// TwinCAT 3 PLC project PRG_PLC
// ProgramVersion: 3.1.4023.0
// CompilerDefines: VISU_USEWSTRING
// libraries:
//   Tc2_Standard, * (Beckhoff Automation GmbH)
//   Tc2_System, * (Beckhoff Automation GmbH)
//   Tc2_Utilities, * (Beckhoff Automation GmbH)
//   Tc3_Module, * (Beckhoff Automation GmbH)
//   VisuDialogs, * (System)
//   VisuSymbols,3.5.10.0,System
// project tree:
//   / GlobalTextList.TcGTLO, ImagePool.TcIPO (not stored), PlcTask.TcTTO, Visualization Manager.TcVMO (not stored), VISU_TASK.TcTTO
//   GVLs/ GVL_Elementy.TcGVL, GVL_Parametry.TcGVL, GVL_Podzespoly.TcGVL, GVL_Wejscia_IO.TcGVL, GVL_Wyjscia_IO.TcGVL
//   POUs/01 - Elementy/Czujnik/ITF/ ITF_Czujnik.TcIO
//   POUs/01 - Elementy/Czujnik/POU/ FB_Czujnik_NC.TcPOU, FB_Czujnik_NO.TcPOU
//   POUs/01 - Elementy/Elektrozawór/ITF/ ITF_Elektozawor.TcIO
//   POUs/01 - Elementy/Elektrozawór/POU/ FB_Elektrozawor_5na2_1Cewka.TcPOU, FB_Elektrozawor_5na2_2Cewki.TcPOU, FB_Elektrozawor_5na3_Odpowietrzony.TcPOU, FB_Elektrozawor_5na3_Zapowietrzony.TcPOU
//   POUs/01 - Elementy/Silownik/DUT/ DUT_SilownikParametry.TcDUT
//   POUs/01 - Elementy/Silownik/ITF/ ITF_Silownik.TcIO
//   POUs/01 - Elementy/Silownik/POU/ FB_Silownik.TcPOU, FB_Silownik_Kontrola.TcPOU, FB_Silownik_Kontrola_Komunikacja.TcPOU
//   POUs/02 - Przesuwacz Na Silowniku/DUT/ DUT_PrzesuwaczNaSilowniku_Parametry.TcDUT (not stored)
//   POUs/02 - Przesuwacz Na Silowniku/POU/ FB_PrzesuwaczNaSilowniku.TcPOU, FB_PrzesuwaczNaSilowniku_Komunikacja.TcPOU (not stored)
//   POUs/03 - Ciecie/DUT/ DUT_Ciecie_Parametry.TcDUT
//   POUs/03 - Ciecie/POU/ FB_Ciecie.TcPOU, FB_Ciecie_Komunikacja.TcPOU
//   POUs/50 - testowy podzespol/POU/ FB_TestowyPodzespol.TcPOU
//   POUs/51 - Krajalnica/DUT/ DUT_Krajalnica_Parametry.TcDUT, DUT_Krajalnica_StanyPodzespolow.TcDUT, DUT_Krajalnica_Symulacja.TcDUT
//   POUs/51 - Krajalnica/POU/ FB_Krajalnica.TcPOU, FB_Krajalnica_Komunikacja.TcPOU
//   POUs/80 - Symulacja pracy/DUT/ DUT_Symulacja_Parametry.TcDUT
//   POUs/80 - Symulacja pracy/POU/ FB_Symulacja.TcPOU
//   POUs/90 - Stan Maszyny/DUT/ DUT_StanMaszyny_VISU_Stan.TcDUT, E_PMLState.TcDUT, E_PMLUnitMode.TcDUT
//   POUs/90 - Stan Maszyny/GVL/ GVL_StanMaszyny.TcGVL, GVL_StanMaszyny_STALE.TcGVL
//   POUs/90 - Stan Maszyny/ITF/ ITF_StanMaszyny.TcIO
//   POUs/90 - Stan Maszyny/POU/ FB_StanMaszyny.TcPOU, FB_StanMaszyny_Baza.TcPOU
//   POUs/90 - Stan Maszyny/Visu/ Visu_StanMaszyny_AktualyStan.TcVIS, Visu_StanMaszyny_AktualyStan_BezNaciskania.TcVIS, Visu_StanMaszyny_Diagram.TcVIS, Visu_StanMaszyny_DiagramZPrzyciskami.TcVIS
//   POUs/91 - Elementy Sterujace/GVL/ GVL_ElementySterujace.TcGVL
//   POUs/91 - Elementy Sterujace/POU/ FB_ElementySterujace.TcPOU
//   POUs/92 - Elementy maszyny/Impulsy/POU/ FB_Impulsy.TcPOU
//   POUs/92 - Elementy maszyny/Przycisk/ITF/ ITF_Przycisk.TcIO
//   POUs/92 - Elementy maszyny/Przycisk/POU/ FB_Przycisk_NC.TcPOU, FB_Przycisk_NO.TcPOU
//   POUs/92 - Elementy maszyny/Wieza Sygnalizacyjna/ITF/ ITF_WiezaSygnalizacyjna.TcIO
//   POUs/92 - Elementy maszyny/Wieza Sygnalizacyjna/POU/ FB_WiezaSygnalizacyjna_Cyfrowe.TcPOU
//   POUs/93 - Podzespol/ITF/ ITF_Podzespol.TcIO
//   POUs/93 - Podzespol/POU/ FB_Podzespol.TcPOU
//   POUs/95 - Logowanie bledow/DUT/ DUT_LogowanieBledow_WyswietlanieParametry.TcDUT, DUT_LogowanieBledow_Zapamietanych.TcDUT, DUT_LogowanieBledow_Zdarzenie.TcDUT, DUT_LogowanieBledow_ZdarzenieOpis.TcDUT, DUT_LogowanieBledow_ZdarzenieStan.TcDUT, DUT_LogowanieBledow_ZdarzenieWyswietlane.TcDUT
//   POUs/95 - Logowanie bledow/GVL/ GVL_LogowanieBledow.TcGVL, GVL_LogowanieBledow_Stale.TcGVL
//   POUs/95 - Logowanie bledow/ITF/ ITF_LogowanieBledow_ElementWykonawczy.TcIO
//   POUs/95 - Logowanie bledow/POU/ FB_LogowanieBledow.TcPOU, FB_LogowanieBledow_ElementWykonawczy.TcPOU, FB_LogowanieBledow_ElementZlozony.TcPOU
//   POUs/95 - Logowanie bledow/Wizualizacja/ Visu_LogowanieBledow_Tabela.TcVIS
//   POUs/99 - Wizualizacja/DUT/ DUT_Wizualizacja_SymulacjaDane.TcDUT
//   POUs/99 - Wizualizacja/GVL/ GVL_Wizualizacja.TcGVL (not stored)
//   POUs/99 - Wizualizacja/POU/ FB_Wizualizacja.TcPOU
//   POUs/ MAIN.TcPOU
//   VISUs/ OknoGlowne.TcVIS, Symulacja.TcVIS, Ustawienia.TcVIS, Visualization.TcVIS
// real-time tasks:
//   TASK PlcTask: cycle T#10ms, priority 20, ADS port 350
//   TASK VISU_TASK: cycle T#200000us, priority 30, ADS port 351

CONFIGURATION PRG_PLC
    RESOURCE PLC ON TwinCAT3
        TASK PlcTask(INTERVAL := T#10ms, PRIORITY := 20);
        TASK VISU_TASK(INTERVAL := T#100us, PRIORITY := 30);
        PROGRAM MAIN WITH PlcTask : MAIN;
        PROGRAM VisuElems_Visu_Prg WITH VISU_TASK : VisuElems.Visu_Prg;
    END_RESOURCE
END_CONFIGURATION

// ---- POUs/01 - Elementy/Silownik/DUT/DUT_SilownikParametry.TcDUT
TYPE DUT_SilownikParametry :
STRUCT
	rCzasNaPrace							: REAL := 5000;
	rCzasNaPowrot							: REAL := 5000;
END_STRUCT
END_TYPE

// ---- POUs/03 - Ciecie/DUT/DUT_Ciecie_Parametry.TcDUT
TYPE DUT_Ciecie_Parametry :
STRUCT
	stNaped									: DUT_SilownikParametry;
	rOdczekaj								: real := 1000; 	//chwila na odczekanie po cięciu
END_STRUCT
END_TYPE

// ---- POUs/51 - Krajalnica/DUT/DUT_Krajalnica_Parametry.TcDUT
TYPE DUT_Krajalnica_Parametry :
STRUCT
	stCiecie1								: DUT_Ciecie_Parametry;	
	stCiecie2								: DUT_Ciecie_Parametry;
	stPodawanieWafla						: DUT_PrzesuwaczNaSilowniku_Parametry;
	
	
END_STRUCT
END_TYPE

// ---- POUs/51 - Krajalnica/DUT/DUT_Krajalnica_StanyPodzespolow.TcDUT
TYPE DUT_Krajalnica_StanyPodzespolow :
STRUCT
	bCiecie1_Bazowanie						: BOOL;
	bCiecie1_Ciecie							: BOOL;
	bCiecie1_Naped_WStronePoczatku			: BOOL;
	bCiecie1_Naped_WStroneKonca				: BOOL;			

	bCiecie2_Bazowanie						: BOOL;
	bCiecie2_Ciecie							: BOOL;
	bCiecie2_Naped_WStronePoczatku			: BOOL;
	bCiecie2_Naped_WStroneKonca				: BOOL;			

	bPodawanie_Bazowanie					: BOOL;
	bPodawanie_Podawanie					: BOOL;
	bPodawanie_Zabierak_WStronePoczatku		: BOOL;
	bPodawanie_zabierak_WStroneKonca		: BOOL;
	bPodawanie_Przesuwanie_WStronePoczatku	: BOOL;
	bPodawanie_Przesuwanie_WStroneKonca		: BOOL;

	
END_STRUCT
END_TYPE

// ---- POUs/51 - Krajalnica/DUT/DUT_Krajalnica_Symulacja.TcDUT
TYPE DUT_Krajalnica_Symulacja :
STRUCT
	bCiecie1Bazuj							: BOOL;		
	bCiecie1Tnij							: BOOL;
	bCiecie2Bazuj							: BOOL;		
	bCiecie2Tnij							: BOOL;
	bPodawanieBazuj							: BOOL;		
	bPodawaniePodaj							: BOOL;	
	
END_STRUCT
END_TYPE

// ---- POUs/80 - Symulacja pracy/DUT/DUT_Symulacja_Parametry.TcDUT
TYPE DUT_Symulacja_Parametry :
STRUCT
	rCiecie1_BazowanieCzasNaPowrot			: REAL := 2000;
	rCiecie1_CiecieCzasNaCiecie				: REAL := 2000;
	rCiecie1_CiecieCzasNaPowrot				: REAL := 2000;
	
	rCiecie2_BazowanieCzasNaPowrot			: REAL := 2000;
	rCiecie2_CiecieCzasNaCiecie				: REAL := 2000;
	rCiecie2_CiecieCzasNaPowrot				: REAL := 2000;
	
	rPodawanieZabierak_BazowanieCzasNaPowrot	: REAL := 1000;
	rPodawaniePrzesuwanie_BazowanieCzasNaPowrot	: REAL := 2000;
	
	rPodawanieZabierak_PodawanieCzasNaPrace			: REAL := 1000;
	rPodawanieZabierak_PodawanieCzasNaPowrot		: REAL := 1000;
	rPodawaniePrzesuwanie_PodawanieCzasNaPobranie	: REAL := 2000;
	rPodawaniePrzesuwanie_PodawanieCzasNaPodanie	: REAL := 2000;
	
END_STRUCT
END_TYPE

// ---- POUs/90 - Stan Maszyny/DUT/DUT_StanMaszyny_VISU_Stan.TcDUT
//==================================================================================================
//								RJM Maszyny sp. z o.o.
//									27.06.2022
//	Struktura sterująca wyświetlania pojedynczego stanu
// 	v1.0	|| TC v 3.1.4024.29		|| - pierwsza wersja
//==================================================================================================
TYPE DUT_StanMaszyny_VISU_Stan :
STRUCT
	bAktywny								: BOOL;
	sNazwa									: STRING;
	dwKolorTla								: DWORD;
	bWygaszone								: BOOL;
END_STRUCT
END_TYPE

// ---- POUs/90 - Stan Maszyny/DUT/E_PMLState.TcDUT
(* states according to PackTags v3.0 *)
//==================================================================================================
//								RJM Maszyny sp. z o.o.
//									27.06.2022
//	Spis dostepnych stanow maszyny
// 	v1.0	|| TC v 3.1.4024.29		|| - pierwsza wersja
//==================================================================================================
{attribute 'qualified_only'}
{attribute 'strict'}
TYPE E_PMLState :
(
	UNDEFINED		:=  0,
	CLEARING 		:=  1,
	STOPPED 		:=  2,
	STARTING 		:=  3,
	IDLE 			:=  4,
	SUSPENDED 		:=  5,
	EXECUTE 		:=  6,
	STOPPING	 	:=  7,
	ABORTING 		:=  8,
	ABORTED 		:=  9,
	HOLDING 		:= 10,
	HELD 			:= 11,
	UNHOLDING 		:= 12,
	SUSPENDING 		:= 13,
	UNSUSPENDING 	:= 14,
	RESETTING 		:= 15,
	COMPLETING 		:= 16,
	COMPLETE	 	:= 17
);
END_TYPE

// ---- POUs/90 - Stan Maszyny/DUT/E_PMLUnitMode.TcDUT
{attribute 'qualified_only'}
{attribute 'strict'}
//==================================================================================================
//								RJM Maszyny sp. z o.o.
//									27.06.2022
//	Spis dostepnych trybow pracy maszyny
// 	v1.0	|| TC v 3.1.4024.29		|| - pierwsza wersja
//==================================================================================================
TYPE E_PMLUnitMode :
(
	UNDEFINED		:=  0,
	AUTOMATIC		:=  1,
	MAINTENANCE 	:=  2,
	MANUAL 			:=  3,
	SEMIAUTOMATIC	:=  4,
	DRYRUN			:=  5,
	USERMODE1		:=  6,
	USERMODE2		:=  7,
	IDLE 			:=  8,
	ESTOP 			:=  9
);
END_TYPE

// ---- POUs/95 - Logowanie bledow/DUT/DUT_LogowanieBledow_WyswietlanieParametry.TcDUT
//==================================================================================================
//								RJM Maszyny sp. z o.o.
//									04.02.2022
//	Struktura parametrów wyświetlania danych historii zdarzeń
// 	v1.0	|| TC v 3.1.4024.22		|| - pierwsza wersja
//==================================================================================================
TYPE DUT_LogowanieBledow_WyswietlanieParametry :
STRUCT
//FILTRY WYSIETLANIA
	// Flagi wykonywalnosci
	bFiltrID								: BOOL;
	bFiltrRodzaj							: BOOL;
	bFiltrStartOD							: BOOL;
	bFiltrStartDO							: BOOL;
	bFiltrKoniecOD							: BOOL;
	bFiltrKoniecDO							: BOOL;
	bFiltrAktywne							: BOOL;
	// Parametry
	iFiltrID								: INT;	
	byFiltrRodzaj							: BYTE;
	dtFiltrStartOD							: DT;
	dtFiltrStartDO							: DT;
	dtFiltrKoniecOD							: DT;
	dtFiltrKoniecDO							: DT;
	
END_STRUCT
END_TYPE

// ---- POUs/95 - Logowanie bledow/DUT/DUT_LogowanieBledow_Zapamietanych.TcDUT
TYPE DUT_LogowanieBledow_Zapamietanych :
STRUCT
	iIdZdarzenia							: INT;
	dtDataStart								: DT;
	dtDataKoniec							: DT;
	bAktywne								: BOOL;
END_STRUCT
END_TYPE

// ---- POUs/95 - Logowanie bledow/DUT/DUT_LogowanieBledow_Zdarzenie.TcDUT
TYPE DUT_LogowanieBledow_Zdarzenie :
STRUCT
	iIdZdarzenia							: INT;
	sNrKomponentu							: STRING[10];
	sKodBledu								: STRING[10];
	byRodzajZdarzenia						: BYTE;	//1 - blad, 2 - ostrzezenie, 3 - wiadomosc, 4 - safety
END_STRUCT
END_TYPE

// ---- POUs/95 - Logowanie bledow/DUT/DUT_LogowanieBledow_ZdarzenieOpis.TcDUT
TYPE DUT_LogowanieBledow_ZdarzenieOpis :
STRUCT
	iIdZdarzenia							: INT;
	sOpis									: STRING;
END_STRUCT
END_TYPE

// ---- POUs/95 - Logowanie bledow/DUT/DUT_LogowanieBledow_ZdarzenieStan.TcDUT
TYPE DUT_LogowanieBledow_ZdarzenieStan :
STRUCT
	iIdZdarzenia							: INT;
	bAktywne								: BOOL;
END_STRUCT
END_TYPE

// ---- POUs/95 - Logowanie bledow/DUT/DUT_LogowanieBledow_ZdarzenieWyswietlane.TcDUT
TYPE DUT_LogowanieBledow_ZdarzenieWyswietlane :
STRUCT
	sNrKomponentu							: STRING[10];
	sKodBledu								: STRING[10];
	byRodzajZdarzenia						: BYTE;
	sOpis									: STRING;
	dtDataStart								: DT;
	dtDataKoniec							: DT;
	dwKolor									: UDINT;
END_STRUCT
END_TYPE

// ---- POUs/99 - Wizualizacja/DUT/DUT_Wizualizacja_SymulacjaDane.TcDUT
TYPE DUT_Wizualizacja_SymulacjaDane :
STRUCT
	stStanySilownikow						: DUT_Krajalnica_StanyPodzespolow;
	eTrybPracy								: E_PMLUnitMode;
	bCiecie1_Poczatek						: BOOL;
	bCiecie1_Koniec							: BOOL;
	bCiecie2_Poczatek						: BOOL;
	bCiecie2_Koniec							: BOOL;
	bPodawanieZabierakPoczatek				: BOOL;
	bPodawanieZabierakKoniec				: BOOL;
	bPodawaniePrzesuwaniePoczatek			: BOOL;
	bPodawaniePrzesuwanieKoniec				: BOOL;
	bCzujnikWaflaDoPodania					: BOOL;
	bCzujnikWaflaDoCiecia1					: BOOL;
	bCzujnikWaflaDoCiecia2					: BOOL;	
	
	bCiecie1Bazuj							: BOOL;
	bCiecie1Tnij							: BOOL;
	bCiecie2Bazuj							: BOOL;		
	bCiecie2Tnij							: BOOL;
	bPodawanieBazuj							: BOOL;		
	bPodawaniePodaj							: BOOL;	

END_STRUCT
END_TYPE

// ---- GVLs/GVL_Elementy.TcGVL
{attribute 'qualified_only'}
{attribute 'global_init_slot' := '40501'}
VAR_GLOBAL
	fbPrzysciskStart						: FB_Przycisk_NO;
	fbPrzyciskStop							: FB_Przycisk_NO;
	fbWieza									: FB_WiezaSygnalizacyjna_Cyfrowe;

END_VAR



	(*
	fbSilownikCiecia1						: FB_Silownik_Kontrola (	fbCzujnikPozycja0 			:= GVL_Wejscia_IO.bCzujnik0C1, 
																		fbCzujnikPozycjaMax 		:= GVL_Wejscia_IO.bCzujnikMaxC1,
																		fbElektrozawor 				:= GVL_Wyjscia_IO.fbElektrozaworC1);

	fbSilownikCiecia2						: FB_Silownik_Kontrola (	fbCzujnikPozycja0 			:= GVL_Wejscia_IO.bCzujnik0C2, 
																		fbCzujnikPozycjaMax 		:= GVL_Wejscia_IO.bCzujnikMaxC2,
																		fbElektrozawor 				:= GVL_Wyjscia_IO.fbElektrozaworC2);

	fbPodawanieWaflaZabierak				: FB_Silownik_Kontrola (	fbCzujnikPozycja0 			:= GVL_Wejscia_IO.bCzujnik0PW_Z, 
																		fbCzujnikPozycjaMax 		:= GVL_Wejscia_IO.bCzujnikMaxPW_Z,
																		fbElektrozawor 				:= GVL_Wyjscia_IO.fbElektrozaworPW_Z);																	
		
	fbPodawanieWaflaPrzesuwanie				: FB_Silownik_Kontrola (	fbCzujnikPozycja0 			:= GVL_Wejscia_IO.bCzujnik0PW_N, 
																		fbCzujnikPozycjaMax 		:= GVL_Wejscia_IO.bCzujnikMaxPW_N,
																		fbElektrozawor 				:= GVL_Wyjscia_IO.fbElektrozaworPW_N);																	

	*)

// ---- GVLs/GVL_Parametry.TcGVL
{attribute 'qualified_only'}
VAR_GLOBAL
	stSymulacja								: DUT_Symulacja_Parametry;
	stKrajalnica							: DUT_Krajalnica_Parametry;
END_VAR

// ---- GVLs/GVL_Podzespoly.TcGVL
{attribute 'qualified_only'}
{attribute 'global_init_slot' := '40505'}
VAR_GLOBAL
	
	fbSymulacja								: FB_Symulacja;	

	fbKrajalnica							: FB_Krajalnica ( 	bC1_Czujnik0					:= GVL_Wejscia_IO.bCzujnik0C1,	
                                                                bC1_CzujnikMax					:= GVL_Wejscia_IO.bCzujnikMaxC1,
                                                                fbC1_Elektrozawor				:= GVL_Wyjscia_IO.fbElektrozaworC1,
																bC2_Czujnik0					:= GVL_Wejscia_IO.bCzujnik0C2,	
                                                                bC2_CzujnikMax					:= GVL_Wejscia_IO.bCzujnikMaxC2,
                                                                fbC2_Elektrozawor				:= GVL_Wyjscia_IO.fbElektrozaworC2,
																bPW_Z_Czujnik0		    		:= GVL_Wejscia_IO.bCzujnik0PW_Z,
																bPW_Z_CzujnikMax	   			:= GVL_Wejscia_IO.bCzujnikMaxPW_Z,
																fbPW_Z_Elektrozawor				:= GVL_Wyjscia_IO.fbElektrozaworPW_Z,
																bPW_P_Czujnik0		    		:= GVL_Wejscia_IO.bCzujnik0PW_N,
																bPW_P_CzujnikMax	   			:= GVL_Wejscia_IO.bCzujnikMaxPW_N,
																fbPW_P_Elektrozawor				:= GVL_Wyjscia_IO.fbElektrozaworPW_N,
																bWafalNaWejsciu					:= GVL_Wejscia_IO.bWafelNaWejsciu,
                                                                bWafalDoCiecia1					:= GVL_Wejscia_IO.bWafelDoCiecia1,
                                                                bWafalDoCiecia2					:= GVL_Wejscia_IO.bWafelDoCiecia2);

															
END_VAR

// ---- GVLs/GVL_Wejscia_IO.TcGVL
{attribute 'qualified_only'}
{attribute 'global_init_slot' := '40501'}
VAR_GLOBAL
//Przyciski	
	
//czujniki siłownika ciecia 1
	bCzujnik0C1								: FB_Czujnik_NO;
	bCzujnikMaxC1							: FB_Czujnik_NO;
//czujniki siłownika ciecia 2
	bCzujnik0C2								: FB_Czujnik_NO;
	bCzujnikMaxC2							: FB_Czujnik_NO;
//czujniki przesuwacza wafla
	bCzujnik0PW_Z							: FB_Czujnik_NO;
	bCzujnikMaxPW_Z							: FB_Czujnik_NO;
	bCzujnik0PW_N							: FB_Czujnik_NO;
	bCzujnikMaxPW_N							: FB_Czujnik_NO;
//czujnik waflae
	bWafelNaWejsciu							: FB_Czujnik_NO;
	bWafelDoCiecia1							: FB_Czujnik_NO;
	bWafelDoCiecia2							: FB_Czujnik_NO;
	
END_VAR

// ---- GVLs/GVL_Wyjscia_IO.TcGVL
{attribute 'qualified_only'}
{attribute 'global_init_slot' := '40510'}
VAR_GLOBAL
//elektrozawor siłownika 1
	fbElektrozaworC1						: FB_Elektrozawor_5na2_2Cewki;
//elektrozawor siłownika 2
	fbElektrozaworC2						: FB_Elektrozawor_5na2_2Cewki;
//elektrozawory przesuwacza
	fbElektrozaworPW_Z						: FB_Elektrozawor_5na2_2Cewki;
	fbElektrozaworPW_N						: FB_Elektrozawor_5na2_2Cewki;
END_VAR

// ---- POUs/90 - Stan Maszyny/GVL/GVL_StanMaszyny.TcGVL
{attribute 'qualified_only'}
{attribute 'global_init_slot' := '40515'}
VAR_GLOBAL

	arrPodzesoly							: ARRAY [1..GVL_StanMaszyny_Stale.MAX_LICZBA_PODZESPOLOW] OF ITF_StanMaszyny :=[
																GVL_Podzespoly.fbSymulacja,
																GVL_Podzespoly.fbKrajalnica];
	fbStanMaszyny							: FB_StanMaszyny (arrPodzesoly := arrPodzesoly,
																iIloscDodanychPodzespolow := 2);
	bStart									: BOOL;
	bStop									: BOOL;
	bReset									: BOOL;
	bAbort									: BOOL;
	bClear									: BOOL;
	bHold									: BOOL;
	bUnhold									: BOOL;
	bSuspend								: BOOL;
	bUnsuspend								: BOOL;
	eTrybPracy								: E_PMLUnitMode := E_PMLUnitMode.MANUAL;		
	bWlaczPrzyciski							: BOOL;												
	
END_VAR

// ---- POUs/90 - Stan Maszyny/GVL/GVL_StanMaszyny_STALE.TcGVL
{attribute 'qualified_only'}
VAR_GLOBAL CONSTANT
	MAX_LICZBA_PODZESPOLOW					: int := 10;
END_VAR

// ---- POUs/91 - Elementy Sterujace/GVL/GVL_ElementySterujace.TcGVL
{attribute 'qualified_only'}
{attribute 'global_init_slot' := '40520'}
VAR_GLOBAL
	fbElementySterujace						: FB_ElementySterujace (
													fbWieza					:= GVL_Elementy.fbWieza,
													fbPrzyciskStart			:= GVL_Elementy.fbPrzysciskStart,
													fbPrzyciskStop			:= GVL_Elementy.fbPrzyciskStop
												);
												
END_VAR

// ---- POUs/95 - Logowanie bledow/GVL/GVL_LogowanieBledow.TcGVL
{attribute 'qualified_only'}
{attribute 'global_init_slot' := '40550'}
VAR_GLOBAL
	arrElementyWykonawcze 					: ARRAY [1..GVL_LogowanieBledow_Stale.MAX_ILOSC_ELEMENTOW] OF 
																ITF_LogowanieBledow_ElementWykonawczy := [
																	GVL_Podzespoly.fbKrajalnica.fbLBKomunikacja];

	fbLoger 								: FB_LogowanieBledow (	tablica := arrElementyWykonawcze,
																	iIloscDodanychElementow := 1);
	bWyswietlAlarmy							: BOOL;																
	
END_VAR
VAR_GLOBAL //PERSISTENT
	arrTablicaZdarzenZapamietancyh			: ARRAY [1..GVL_LogowanieBledow_Stale.MAX_ILOSC_ZDARZEN_ZAPAMIETANYCH] OF DUT_LogowanieBledow_Zapamietanych;																
	
	iIloscZdarzenZapamietanych				: INT;	//ilosc zdarzen ktore wystapiły
END_VAR

// ---- POUs/95 - Logowanie bledow/GVL/GVL_LogowanieBledow_Stale.TcGVL
{attribute 'qualified_only'}
VAR_GLOBAL CONSTANT
	MAX_ILOSC_ELEMENTOW						: INT := 10;	//Ilosc elementow zlozonych
	MAX_ILOSC_ZDARZEN_NA_ELEMENT			: INT := 10;	//ilosc zdarzen na element
	MAX_ILOSC_ELEMENTOW_NA_PODZESPOL		: INT := 10;	//Ilosc elementow na element złozony
	MAX_ILOSC_ZDARZEN						: INT := 100;	//ilosc zdarzen zdefiniowanych
	MAX_ILOSC_ZDARZEN_DO_WYSWIETLANIA		: INT := 50;	//ilosc wyswietlanych zdarzen z tablicy zapamietanych
	MAX_ILOSC_ZDARZEN_ZAPAMIETANYCH			: INT := 200;	//ilosc zadarzen zapamietanych
END_VAR

// ---- POUs/01 - Elementy/Czujnik/ITF/ITF_Czujnik.TcIO
//==================================================================================================
//								RJM Maszyny sp. z o.o.
//									04.06.2022
//	Obsługa czujnika  
// 	v1.0	|| TC v 3.1.4024.22		|| - pierwsza wersja
//==================================================================================================
INTERFACE ITF_Czujnik

//==================================================================================================
//								RJM Maszyny sp. z o.o.
//									13.05.2022
//	Informacja czy czujnik jest zadziałany 
// 	v1.0	|| TC v 3.1.4024.22		|| - pierwsza wersja
//==================================================================================================
PROPERTY CzyZadzialany : BOOL
GET
END_GET
END_PROPERTY

END_INTERFACE

// ---- POUs/01 - Elementy/Elektrozawór/ITF/ITF_Elektozawor.TcIO
//==================================================================================================
//								RJM Maszyny sp. z o.o.
//									04.06.2022
//	Sterowanie elektrozaworem  
// 	v1.0	|| TC v 3.1.4024.22		|| - pierwsza wersja
//==================================================================================================
INTERFACE ITF_Elektozawor

//==================================================================================================
//								RJM Maszyny sp. z o.o.
//									04.06.2022
//	Sterowanie cewkami elektrozaworu 
// 	v1.0	|| TC v 3.1.4024.22		|| - pierwsza wersja
//==================================================================================================
METHOD Steruj : BOOL
VAR_INPUT
	bKierunekWstrone0						: BOOL;
	bKierunekWStroneMax						: BOOL;	
END_VAR
END_METHOD

END_INTERFACE

// ---- POUs/01 - Elementy/Silownik/ITF/ITF_Silownik.TcIO
//==================================================================================================
//								RJM Maszyny sp. z o.o.
//									13.05.2022
//	Obsługa silonwika
// 	v1.0	|| TC v 3.1.4024.22		|| - pierwsza wersja
//==================================================================================================
INTERFACE ITF_Silownik

//==================================================================================================
//								RJM Maszyny sp. z o.o.
//									13.05.2022
//	Informaca czy  tłoczysko jest na końca
// 	v1.0	|| TC v 3.1.4024.22		|| - pierwsza wersja
//==================================================================================================
PROPERTY NaKoncu : BOOL
GET
END_GET
END_PROPERTY

//==================================================================================================
//								RJM Maszyny sp. z o.o.
//									13.05.2022
//	Informaca czy  tłoczysko jest na poczatku
// 	v1.0	|| TC v 3.1.4024.22		|| - pierwsza wersja
//==================================================================================================
PROPERTY NaPoczatku : BOOL
GET
END_GET
END_PROPERTY

//==================================================================================================
//								RJM Maszyny sp. z o.o.
//									13.05.2022
//	Przesun tłoczysko w strone końca
// 	v1.0	|| TC v 3.1.4024.22		|| - pierwsza wersja
//==================================================================================================
PROPERTY PrzesunDoKonca : BOOL
SET
END_SET
END_PROPERTY

//==================================================================================================
//								RJM Maszyny sp. z o.o.
//									13.05.2022
//	Przesun tłoczysko w strone poczatku
// 	v1.0	|| TC v 3.1.4024.22		|| - pierwsza wersja
//==================================================================================================
PROPERTY PrzesunDoPoczatku : BOOL
SET
END_SET
END_PROPERTY

//==================================================================================================
//								RJM Maszyny sp. z o.o.
//									13.05.2022
//	Przesuwanie tłoczyska w strone końca
// 	v1.0	|| TC v 3.1.4024.22		|| - pierwsza wersja
//==================================================================================================
PROPERTY PrzesuwanieWStroneKonca : BOOL
GET
END_GET
END_PROPERTY

//==================================================================================================
//								RJM Maszyny sp. z o.o.
//									13.05.2022
//	Przesuwanie tłoczyska w strone poczatku
// 	v1.0	|| TC v 3.1.4024.22		|| - pierwsza wersja
//==================================================================================================
PROPERTY PrzesuwanieWStronePoczatku : BOOL
GET
END_GET
END_PROPERTY

END_INTERFACE

// ---- POUs/90 - Stan Maszyny/ITF/ITF_StanMaszyny.TcIO
INTERFACE ITF_StanMaszyny

//==================================================================================================
//								RJM Maszyny sp. z o.o.
//									5.06.2022
//	Stan maszyny Aborted - metoda pusta
// 	v1.0	|| TC v 3.1.4024.29		|| - pierwsza wersja
//==================================================================================================
METHOD SM_Aborted : BOOL
VAR_INPUT
	
END_VAR
END_METHOD

//==================================================================================================
//								RJM Maszyny sp. z o.o.
//									5.06.2022
//	Stan maszyny Aborting - awaryjne zatrzymanie maszyny E-STOP
// 	v1.0	|| TC v 3.1.4024.29		|| - pierwsza wersja
//==================================================================================================
METHOD SM_Aborting : BOOL
VAR_INPUT
END_VAR
END_METHOD

//==================================================================================================
//								RJM Maszyny sp. z o.o.
//									5.06.2022
//	Stan maszyny Clearing
// 	v1.0	|| TC v 3.1.4024.29		|| - pierwsza wersja
//==================================================================================================
METHOD SM_Clearing : BOOL
VAR_INPUT
END_VAR
END_METHOD

//==================================================================================================
//								RJM Maszyny sp. z o.o.
//									5.06.2022
//	Stan maszyny Complete 
// 	v1.0	|| TC v 3.1.4024.29		|| - pierwsza wersja
//==================================================================================================
METHOD SM_Complete : BOOL
VAR_INPUT
END_VAR
END_METHOD

//==================================================================================================
//								RJM Maszyny sp. z o.o.
//									5.06.2022
//	Stan maszyny Completing
// 	v1.0	|| TC v 3.1.4024.29		|| - pierwsza wersja
//==================================================================================================
METHOD SM_Completing : BOOL
VAR_INPUT
END_VAR
END_METHOD

//==================================================================================================
//								RJM Maszyny sp. z o.o.
//									5.06.2022
//	Stan maszyny Execute
// 	v1.0	|| TC v 3.1.4024.29		|| - pierwsza wersja
//==================================================================================================
METHOD SM_Execute : BOOL
VAR_INPUT
	eTrybPracy								: E_PMLUnitMode;
END_VAR
END_METHOD

//==================================================================================================
//								RJM Maszyny sp. z o.o.
//									5.06.2022
//	Stan maszyny Held  - metoda pusta
// 	v1.0	|| TC v 3.1.4024.29		|| - pierwsza wersja
//==================================================================================================
METHOD SM_Held : BOOL
VAR_INPUT
END_VAR
END_METHOD

//==================================================================================================
//								RJM Maszyny sp. z o.o.
//									5.06.2022
//	Stan maszyny Holding
// 	v1.0	|| TC v 3.1.4024.29		|| - pierwsza wersja
//==================================================================================================
METHOD SM_Holding : BOOL
VAR_INPUT
END_VAR
END_METHOD

//==================================================================================================
//								RJM Maszyny sp. z o.o.
//									5.06.2022
//	Stan maszyny Idle
// 	v1.0	|| TC v 3.1.4024.29		|| - pierwsza wersja
//==================================================================================================
METHOD SM_Idle : BOOL
VAR_INPUT
END_VAR
END_METHOD

//==================================================================================================
//								RJM Maszyny sp. z o.o.
//									5.06.2022
//	Stan maszyny Reseting - konczenie niedokocznonych cykli i powrot podzespolami do pozycji startowej
// 	v1.0	|| TC v 3.1.4024.29		|| - pierwsza wersja
//==================================================================================================
METHOD SM_Resetting : BOOL
VAR_INPUT
	eTrybPracy								: E_PMLUnitMode;
END_VAR
END_METHOD

//==================================================================================================
//								RJM Maszyny sp. z o.o.
//									5.06.2022
//	Stan maszyny Starting - Ustawienie elementów do pracy 
// 	v1.0	|| TC v 3.1.4024.29		|| - pierwsza wersja
//==================================================================================================
METHOD SM_Starting : BOOL
VAR_INPUT
END_VAR
END_METHOD

//==================================================================================================
//								RJM Maszyny sp. z o.o.
//									5.06.2022
//	Stan maszyny Stoped - metoda pusta
// 	v1.0	|| TC v 3.1.4024.29		|| - pierwsza wersja
//==================================================================================================
METHOD SM_Stopped : BOOL
VAR_INPUT
END_VAR
END_METHOD

//==================================================================================================
//								RJM Maszyny sp. z o.o.
//									5.06.2022
//	Stan maszyny Stopping - Zakonczenie aktualnych operacji nie zaczynamy kolejnych
// 	v1.0	|| TC v 3.1.4024.29		|| - pierwsza wersja
//==================================================================================================
METHOD SM_Stopping : BOOL
VAR_INPUT
END_VAR
END_METHOD

//==================================================================================================
//								RJM Maszyny sp. z o.o.
//									5.06.2022
//	Stan maszyny Suspended - metoda pusta
// 	v1.0	|| TC v 3.1.4024.29		|| - pierwsza wersja
//==================================================================================================
METHOD SM_Suspended : BOOL
VAR_INPUT
END_VAR
END_METHOD

//==================================================================================================
//								RJM Maszyny sp. z o.o.
//									5.06.2022
//	Stan maszyny Suspending
// 	v1.0	|| TC v 3.1.4024.29		|| - pierwsza wersja
//==================================================================================================
METHOD SM_Suspending : BOOL
VAR_INPUT
END_VAR
END_METHOD

//==================================================================================================
//								RJM Maszyny sp. z o.o.
//									5.06.2022
//	Stan maszyny Unholding
// 	v1.0	|| TC v 3.1.4024.29		|| - pierwsza wersja
//==================================================================================================
METHOD SM_Unholding : BOOL
VAR_INPUT
END_VAR
END_METHOD

//==================================================================================================
//								RJM Maszyny sp. z o.o.
//									5.06.2022
//	Stan maszyny Unsuspending
// 	v1.0	|| TC v 3.1.4024.29		|| - pierwsza wersja
//==================================================================================================
METHOD SM_Unsuspending : BOOL
VAR_INPUT
END_VAR
END_METHOD

END_INTERFACE

// ---- POUs/92 - Elementy maszyny/Przycisk/ITF/ITF_Przycisk.TcIO
INTERFACE ITF_Przycisk

PROPERTY CzyNacisniety : BOOL
GET
END_GET
END_PROPERTY

PROPERTY Podswietlenie : BOOL
SET
END_SET
END_PROPERTY

END_INTERFACE

// ---- POUs/92 - Elementy maszyny/Wieza Sygnalizacyjna/ITF/ITF_WiezaSygnalizacyjna.TcIO
INTERFACE ITF_WiezaSygnalizacyjna

//==================================================================================================
//								RJM Maszyny sp. z o.o.
//									22.06.2022
//	Wlaczanie/Wylaczenia segment bialy   
// 	v1.0	|| TC v 3.1.4024.29		|| - pierwsza wersja
//==================================================================================================
PROPERTY Bialy : BOOL
GET
END_GET
SET
END_SET
END_PROPERTY

//==================================================================================================
//								RJM Maszyny sp. z o.o.
//									22.06.2022
//	Wlaczanie/Wylaczenia segment czerwony   
// 	v1.0	|| TC v 3.1.4024.29		|| - pierwsza wersja
//==================================================================================================
PROPERTY Czerwony : BOOL
GET
END_GET
SET
END_SET
END_PROPERTY

//==================================================================================================
//								RJM Maszyny sp. z o.o.
//									22.06.2022
//	Wlaczanie/Wylaczenia segment niebieski   
// 	v1.0	|| TC v 3.1.4024.29		|| - pierwsza wersja
//==================================================================================================
PROPERTY Niebieski : BOOL
GET
END_GET
SET
END_SET
END_PROPERTY

//==================================================================================================
//								RJM Maszyny sp. z o.o.
//									22.06.2022
//	Wlaczanie/Wylaczenia segment zielony  
// 	v1.0	|| TC v 3.1.4024.29		|| - pierwsza wersja
//==================================================================================================
PROPERTY Zielony : BOOL
GET
END_GET
SET
END_SET
END_PROPERTY

//==================================================================================================
//								RJM Maszyny sp. z o.o.
//									22.06.2022
//	Wlaczanie/Wylaczenia segment zolty   
// 	v1.0	|| TC v 3.1.4024.29		|| - pierwsza wersja
//==================================================================================================
PROPERTY Zolty : BOOL
GET
END_GET
SET
END_SET
END_PROPERTY

END_INTERFACE

// ---- POUs/93 - Podzespol/ITF/ITF_Podzespol.TcIO
INTERFACE ITF_Podzespol

PROPERTY Bazowanie : BOOL
GET
END_GET
END_PROPERTY

PROPERTY Bazuj : BOOL
SET
END_SET
END_PROPERTY

METHOD CyklBazowania_Praca : BOOL
VAR_INPUT
END_VAR
END_METHOD

PROPERTY CyklPracy : BOOL
GET
END_GET
END_PROPERTY

METHOD CyklPracy_Praca : BOOL
VAR_INPUT
END_VAR
END_METHOD

PROPERTY CyklPracySkonczony : BOOL
GET
END_GET
END_PROPERTY

METHOD Praca : BOOL
VAR_INPUT
END_VAR
END_METHOD

METHOD Resetowanie : BOOL
VAR_INPUT
END_VAR
END_METHOD

PROPERTY Resetuj : BOOL
SET
END_SET
END_PROPERTY

PROPERTY WykonajCyklPracy : BOOL
SET
END_SET
END_PROPERTY

END_INTERFACE

// ---- POUs/95 - Logowanie bledow/ITF/ITF_LogowanieBledow_ElementWykonawczy.TcIO
INTERFACE ITF_LogowanieBledow_ElementWykonawczy

METHOD DefinicjaTabeliZdarzen_1031_Niemiecki : BOOL
VAR_INPUT
	arrTablicaDefinicjiZdarzenOpis			: REFERENCE TO ARRAY [1..GVL_LogowanieBledow_Stale.MAX_ILOSC_ZDARZEN] OF DUT_LogowanieBledow_ZdarzenieOpis;

END_VAR
END_METHOD

METHOD DefinicjaTabeliZdarzen_1033_Angielski : BOOL
VAR_INPUT
	arrTablicaDefinicjiZdarzenOpis			: REFERENCE TO ARRAY [1..GVL_LogowanieBledow_Stale.MAX_ILOSC_ZDARZEN] OF DUT_LogowanieBledow_ZdarzenieOpis;

END_VAR
END_METHOD

METHOD DefinicjaTabeliZdarzen_1045_Polski : BOOL
VAR_INPUT
	arrTablicaDefinicjiZdarzenOpis			: REFERENCE TO ARRAY [1..GVL_LogowanieBledow_Stale.MAX_ILOSC_ZDARZEN] OF DUT_LogowanieBledow_ZdarzenieOpis;

END_VAR
END_METHOD

METHOD DefinicjaTabeliZdarzen_Ogolna : BOOL
VAR_INPUT
	arrTablicaDefinicjiZdarzen				: REFERENCE TO ARRAY [1..GVL_LogowanieBledow_Stale.MAX_ILOSC_ZDARZEN] OF DUT_LogowanieBledow_Zdarzenie;
	arrTablicaDefinicjiZdarzenOpis			: REFERENCE TO ARRAY [1..GVL_LogowanieBledow_Stale.MAX_ILOSC_ZDARZEN] OF DUT_LogowanieBledow_ZdarzenieOpis;
	arrTablicaDefinicjiZdarzenStan			: REFERENCE TO ARRAY [1..GVL_LogowanieBledow_Stale.MAX_ILOSC_ZDARZEN] OF DUT_LogowanieBledow_ZdarzenieStan;

	iIdZdarzenia							: REFERENCE TO INT;
	iNrPodzespolu							: INT := 0;
	iNrPodelementu							: INT := 0;
	iNrElementu								: INT := 0;
END_VAR
END_METHOD

METHOD GenerujNrKomponentu : STRING
VAR_INPUT
	iNrPodzespolu							: INT := 0;
	iNrPodelementu							: INT := 0;
	iNrElementu								: INT := 0;
END_VAR
END_METHOD

METHOD ZwrocTabliceDefinicji : BOOL
VAR_INPUT
	arrTablicaDefinicjiZdarzen				: REFERENCE TO ARRAY [1..GVL_LogowanieBledow_Stale.MAX_ILOSC_ZDARZEN] OF DUT_LogowanieBledow_Zdarzenie;
	arrTablicaDefinicjiZdarzenOpis			: REFERENCE TO ARRAY [1..GVL_LogowanieBledow_Stale.MAX_ILOSC_ZDARZEN] OF DUT_LogowanieBledow_ZdarzenieOpis;
	arrTablicaDefinicjiZdarzenStan			: REFERENCE TO ARRAY [1..GVL_LogowanieBledow_Stale.MAX_ILOSC_ZDARZEN] OF DUT_LogowanieBledow_ZdarzenieStan;
	
	iIdZdarzenia							: REFERENCE TO INT;
	iNrPodzespolu							: INT;
	iNrPodelementu							: INT;
	iNrElementu								: INT;
	iJezykId								: INT;
END_VAR
END_METHOD

METHOD ZwrocTabliceStanu : BOOL
VAR_INPUT
	arrTablicaDefinicjiZdarzenStan			: REFERENCE TO ARRAY [1..GVL_LogowanieBledow_Stale.MAX_ILOSC_ZDARZEN] OF DUT_LogowanieBledow_ZdarzenieStan;
END_VAR
END_METHOD

END_INTERFACE

// ---- POUs/MAIN.TcPOU
PROGRAM MAIN
VAR
	bKonfiguruj								: BOOL := TRUE;
	
	fbWizualizacja							: FB_Wizualizacja;
	
END_VAR

IF (bKonfiguruj) THEN
	A_Konfiguracja ();
	bKonfiguruj								:= FALSE;
END_IF
//--------LOGER
	GVL_LogowanieBledow.fbLoger (arrZdarzeniaPamietane 		:= GVL_LogowanieBledow.arrTablicaZdarzenZapamietancyh,
								iIloscZdarzenZapamietanych 	:= GVL_LogowanieBledow.iIloscZdarzenZapamietanych,
								bWyswietlanieTablicyAlarmow	:= GVL_LogowanieBledow.bWyswietlAlarmy);
//--------LOGER
//--------STEROWANIE MASZYNĄ
GVL_StanMaszyny.fbStanMaszyny(
	bStart				:= GVL_StanMaszyny.bStart OR GVL_ElementySterujace.fbElementySterujace.NacisnietyStart, 
	bStop				:= GVL_StanMaszyny.bStop OR GVL_ElementySterujace.fbElementySterujace.NacisnietyStop, 
	bReset				:= GVL_StanMaszyny.bReset, 
	bAbort				:= GVL_StanMaszyny.bAbort, 
	bClear				:= GVL_StanMaszyny.bClear, 
	bHold				:= GVL_StanMaszyny.bHold, 
	bUnHold				:= GVL_StanMaszyny.bUnhold, 
	bSuspend			:= GVL_StanMaszyny.bSuspend, 
	bUnsuspend			:= GVL_StanMaszyny.bUnsuspend,
	eTryb				:= GVL_StanMaszyny.eTrybPracy);


GVL_ElementySterujace.fbElementySterujace ();
GVL_ElementySterujace.fbElementySterujace.StanMaszyny	:= GVL_StanMaszyny.fbStanMaszyny.StanPracy;
GVL_ElementySterujace.fbElementySterujace.TrybPracy		:= GVL_StanMaszyny.fbStanMaszyny.TrybPracy;
//--------STEROWANIE MASZYNĄ

GVL_Podzespoly.fbSymulacja(
								stParametry						:= GVL_Parametry.stSymulacja, 
								stStanyPodzespolow				:= GVL_Podzespoly.fbKrajalnica.stStanyPodzespolow,
								eTrybPracy						:= GVL_StanMaszyny.fbStanMaszyny.TrybPracy, 
								bCiecie1_Poczatek				=> GVL_Wejscia_IO.bCzujnik0C1.bSymulacja, 
								bCiecie1_Koniec					=> GVL_Wejscia_IO.bCzujnikMaxC1.bSymulacja, 
								bCiecie2_Poczatek				=> GVL_Wejscia_IO.bCzujnik0C2.bSymulacja, 
								bCiecie2_Koniec					=> GVL_Wejscia_IO.bCzujnikMaxC2.bSymulacja, 
								bPodawanieZabierakPoczatek		=> GVL_Wejscia_IO.bCzujnik0PW_Z.bSymulacja, 
								bPodawanieZabierakKoniec		=> GVL_Wejscia_IO.bCzujnikMaxPW_Z.bSymulacja, 
								bPodawaniePrzesuwaniePoczatek	=> GVL_Wejscia_IO.bCzujnik0PW_N.bSymulacja, 
								bPodawaniePrzesuwanieKoniec		=> GVL_Wejscia_IO.bCzujnikMaxPW_N.bSymulacja, 
								bCzujnikWaflaDoPodania			=> GVL_Wejscia_IO.bWafelNaWejsciu.bSymulacja, 
								bCzujnikWaflaDoCiecia1			=> GVL_Wejscia_IO.bWafelDoCiecia1.bSymulacja, 
								bCzujnikWaflaDoCiecia2			=> GVL_Wejscia_IO.bWafelDoCiecia2.bSymulacja);
								
GVL_Podzespoly.fbKrajalnica (	stParametry 					:= GVL_Parametry.stKrajalnica,
								stSterowanieSymulacja			:= fbWizualizacja.stSterowanie);

	
fbWizualizacja(
								stStanySilownikow				:= GVL_Podzespoly.fbKrajalnica.stStanyPodzespolow,
								eTrybPracy						:= GVL_StanMaszyny.fbStanMaszyny.TrybPracy,   
								bCiecie1_Poczatek				:= GVL_Wejscia_IO.bCzujnik0C1.CzyZadzialany, 
								bCiecie1_Koniec					:= GVL_Wejscia_IO.bCzujnikMaxC1.CzyZadzialany, 
								bCiecie2_Poczatek				:= GVL_Wejscia_IO.bCzujnik0C2.CzyZadzialany, 
								bCiecie2_Koniec					:= GVL_Wejscia_IO.bCzujnikMaxC2.CzyZadzialany, 
								bPodawanieZabierakPoczatek		:= GVL_Wejscia_IO.bCzujnik0PW_Z.CzyZadzialany, 
								bPodawanieZabierakKoniec		:= GVL_Wejscia_IO.bCzujnikMaxPW_Z.CzyZadzialany, 
								bPodawaniePrzesuwaniePoczatek	:= GVL_Wejscia_IO.bCzujnik0PW_N.CzyZadzialany,
								bPodawaniePrzesuwanieKoniec		:= GVL_Wejscia_IO.bCzujnikMaxPW_N.CzyZadzialany, 
								bCzujnikWaflaDoPodania			:= GVL_Wejscia_IO.bWafelNaWejsciu.CzyZadzialany, 
								bCzujnikWaflaDoCiecia1			:= GVL_Wejscia_IO.bWafelDoCiecia1.CzyZadzialany, 
								bCzujnikWaflaDoCiecia2			:= GVL_Wejscia_IO.bWafelDoCiecia2.CzyZadzialany);

ACTION A_Konfiguracja:
	GVL_StanMaszyny.fbStanMaszyny.KonfiguracjaStanowPracyDlaTrybu(
		eNrTrybu		:= E_PMLUnitMode.AUTOMATIC,  
		bClearing		:= TRUE, 
		bStopped		:= TRUE, 
		bStarting		:= TRUE, 
		bIdle			:= TRUE, 
		bSuspended		:= TRUE, 
		bExecute		:= TRUE, 
		bStopping		:= TRUE, 
		bAborting		:= TRUE, 
		bAborted		:= TRUE, 
		bHolding		:= TRUE, 
		bHeld			:= TRUE, 
		bUnholding		:= TRUE, 
		bSuspending		:= TRUE, 
		bUnsuspending	:= TRUE, 
		bResetting		:= TRUE, 
		bCompleting		:= TRUE, 
		bComplete		:= TRUE);
	GVL_StanMaszyny.fbStanMaszyny.KonfiguracjaStanowPracyDlaTrybu(
		eNrTrybu		:= E_PMLUnitMode.MANUAL, 
		bClearing		:= TRUE, 
		bStopped		:= TRUE, 
		bStarting		:= TRUE, 
		bIdle			:= TRUE, 
		bSuspended		:= FALSE, 
		bExecute		:= TRUE, 
		bStopping		:= TRUE, 
		bAborting		:= TRUE, 
		bAborted		:= TRUE, 
		bHolding		:= FALSE, 
		bHeld			:= FALSE, 
		bUnholding		:= FALSE, 
		bSuspending		:= FALSE, 
		bUnsuspending	:= FALSE, 
		bResetting		:= TRUE, 
		bCompleting		:= FALSE, 
		bComplete		:= FALSE);
	GVL_StanMaszyny.fbStanMaszyny.KonfiguracjaStanowPracyDlaTrybu(
		eNrTrybu		:= E_PMLUnitMode.SEMIAUTOMATIC, 
		bClearing		:= TRUE, 
		bStopped		:= TRUE, 
		bStarting		:= TRUE, 
		bIdle			:= TRUE, 
		bSuspended		:= FALSE, 
		bExecute		:= TRUE, 
		bStopping		:= TRUE, 
		bAborting		:= TRUE, 
		bAborted		:= TRUE, 
		bHolding		:= FALSE, 
		bHeld			:= FALSE, 
		bUnholding		:= FALSE, 
		bSuspending		:= FALSE, 
		bUnsuspending	:= FALSE, 
		bResetting		:= TRUE, 
		bCompleting		:= FALSE, 
		bComplete		:= FALSE);
END_ACTION

END_PROGRAM

// ---- POUs/99 - Wizualizacja/POU/FB_Wizualizacja.TcPOU
FUNCTION_BLOCK FB_Wizualizacja
VAR_INPUT
	stStanySilownikow						: DUT_Krajalnica_StanyPodzespolow;
	eTrybPracy								: E_PMLUnitMode;
	bCiecie1_Poczatek						: BOOL;
	bCiecie1_Koniec							: BOOL;
	bCiecie2_Poczatek						: BOOL;
	bCiecie2_Koniec							: BOOL;
	bPodawanieZabierakPoczatek				: BOOL;
	bPodawanieZabierakKoniec				: BOOL;
	bPodawaniePrzesuwaniePoczatek			: BOOL;
	bPodawaniePrzesuwanieKoniec				: BOOL;
	bCzujnikWaflaDoPodania					: BOOL;
	bCzujnikWaflaDoCiecia1					: BOOL;
	bCzujnikWaflaDoCiecia2					: BOOL;
END_VAR
VAR_OUTPUT
	stSterowanie							: DUT_Krajalnica_Symulacja;
END_VAR
VAR
	stDane									: DUT_Wizualizacja_SymulacjaDane;
END_VAR

stDane.stStanySilownikow					:= stStanySilownikow;
stDane.eTrybPracy							:= eTrybPracy;
stDane.bCiecie1_Poczatek					:= bCiecie1_Poczatek;				         
stDane.bCiecie1_Koniec						:= bCiecie1_Koniec;					          
stDane.bCiecie2_Poczatek					:= bCiecie2_Poczatek;				         
stDane.bCiecie2_Koniec						:= bCiecie2_Koniec;					          
stDane.bPodawanieZabierakPoczatek			:= bPodawanieZabierakPoczatek;		  
stDane.bPodawanieZabierakKoniec		    	:= bPodawanieZabierakKoniec;		    
stDane.bPodawaniePrzesuwaniePoczatek		:= bPodawaniePrzesuwaniePoczatek;	
stDane.bPodawaniePrzesuwanieKoniec			:= bPodawaniePrzesuwanieKoniec;		 
stDane.bCzujnikWaflaDoPodania				:= bCzujnikWaflaDoPodania;			     
stDane.bCzujnikWaflaDoCiecia1				:= bCzujnikWaflaDoCiecia1;			     
stDane.bCzujnikWaflaDoCiecia2				:= bCzujnikWaflaDoCiecia2;

stSterowanie.bCiecie1Bazuj					:= stDane.bCiecie1Bazuj;
stSterowanie.bCiecie1Tnij					:= stDane.bCiecie1Tnij;

END_FUNCTION_BLOCK

// ---- POUs/92 - Elementy maszyny/Przycisk/POU/FB_Przycisk_NO.TcPOU
//==================================================================================================
//								RJM Maszyny sp. z o.o.
//									22.06.2022
//	Obsługa przycisku ze stykiem NO
// 	v1.0	|| TC v 3.1.4024.22		|| - pierwsza wersja
//==================================================================================================
FUNCTION_BLOCK FB_Przycisk_NO IMPLEMENTS ITF_Przycisk
VAR
	bStyk							AT %I*	: BOOL;
	bPodswietlenie					AT %Q*	: BOOL;
END_VAR

PROPERTY CzyNacisniety : BOOL
GET
CzyNacisniety								:= bStyk;
END_GET
END_PROPERTY

PROPERTY Podswietlenie : BOOL
SET
bPodswietlenie								:= Podswietlenie;
END_SET
END_PROPERTY

END_FUNCTION_BLOCK

// ---- POUs/92 - Elementy maszyny/Wieza Sygnalizacyjna/POU/FB_WiezaSygnalizacyjna_Cyfrowe.TcPOU
FUNCTION_BLOCK FB_WiezaSygnalizacyjna_Cyfrowe IMPLEMENTS ITF_WiezaSygnalizacyjna
VAR
	bCzerwony						AT%Q*	: BOOL;
	bZolty							AT%Q*	: BOOL;
	bZielony						AT%Q*	: BOOL;
	bNiebieski						AT%Q*	: BOOL;
	bBialy							AT%Q*	: BOOL;
	
END_VAR

(*==================================================================================================
								RJM Maszyny sp. z o.o.
									22.06.2022
	Wlaczanie/Wylaczenia segment bialy   
 	v1.0	|| TC v 3.1.4024.29		|| - pierwsza wersja
==================================================================================================*)
PROPERTY Bialy : BOOL
GET
Bialy										:= bBialy;
END_GET
SET
bBialy										:= Bialy;
END_SET
END_PROPERTY

(*==================================================================================================
								RJM Maszyny sp. z o.o.
									22.06.2022
	Wlaczanie/Wylaczenia segment czerwony   
 	v1.0	|| TC v 3.1.4024.29		|| - pierwsza wersja
==================================================================================================*)
PROPERTY Czerwony : BOOL
GET
Czerwony									:= bCzerwony;
END_GET
SET
bCzerwony									:= Czerwony;
END_SET
END_PROPERTY

(*==================================================================================================
								RJM Maszyny sp. z o.o.
									22.06.2022
	Wlaczanie/Wylaczenia segment niebieski   
 	v1.0	|| TC v 3.1.4024.29		|| - pierwsza wersja
==================================================================================================*)
PROPERTY Niebieski : BOOL
GET
Niebieski									:= bNiebieski;
END_GET
SET
bNiebieski									:= Niebieski;
END_SET
END_PROPERTY

(*==================================================================================================
								RJM Maszyny sp. z o.o.
									22.06.2022
	Wlaczanie/Wylaczenia segment zielony  
 	v1.0	|| TC v 3.1.4024.29		|| - pierwsza wersja
==================================================================================================*)
PROPERTY Zielony : BOOL
GET
Zielony										:= bZielony;
END_GET
SET
bZielony									:= Zielony;
END_SET
END_PROPERTY

(*==================================================================================================
								RJM Maszyny sp. z o.o.
									22.06.2022
	Wlaczanie/Wylaczenia segment zolty   
 	v1.0	|| TC v 3.1.4024.29		|| - pierwsza wersja
==================================================================================================*)
PROPERTY Zolty : BOOL
GET
Zolty										:= bZolty;
END_GET
SET
bZolty										:= Zolty;
END_SET
END_PROPERTY

END_FUNCTION_BLOCK

// ---- POUs/01 - Elementy/Silownik/POU/FB_Silownik_Kontrola.TcPOU
//==================================================================================================
//								RJM Maszyny sp. z o.o.
//									13.05.2022
//	Obsługa silonwika podstawa z kontrolą czasów oraz kontrolą czujników
//	Realizacja wysuwania i chowania tłoczyska dla jednej cewki zwrócenie pozycji skrajnych
// 	v1.0	|| TC v 3.1.4024.22		|| - pierwsza wersja
//==================================================================================================
FUNCTION_BLOCK FB_Silownik_Kontrola EXTENDS FB_Silownik 
VAR_INPUT
	stParametry								: DUT_SilownikParametry;
END_VAR
VAR_OUTPUT
END_VAR
VAR
	tonCzasNaPrace							: TON;
	tonCzasNaPowrot							: TON;
	fbKontrolaCzujnik0_F					: F_TRIG;
	fbKontrolaCzujnikMax_F					: F_TRIG;
	fbKontrolaCzujnik0_R					: R_TRIG;
	fbKontrolaCzujnikMax_R					: R_TRIG;
	fbLBKomunikacja							: FB_Silownik_Kontrola_Komunikacja;
END_VAR

METHOD Praca : BOOL
VAR_INPUT
END_VAR
SUPER^.Praca ();
//Czasy sprawdzające czas wysunięcia lub chowania tłoczyska
	tonCzasNaPrace (IN := bPrzesuwanieWStroneKonca, PT := REAL_TO_TIME (stParametry.rCzasNaPrace));
	tonCzasNaPowrot (In := bPrzesuwanieWStronePoczatku, PT := REAL_TO_TIME (stParametry.rCzasNaPowrot));
//kontrola wysuwania
	IF (tonCzasNaPrace.Q) THEN
		fbLBKomunikacja.UstawStan (iId := 1, bStan := TRUE);
	ELSIF (fbCzujnikPozycjaMax.CzyZadzialany AND NOT bPrzesuwanieWStroneKonca) THEN
		fbLBKomunikacja.UstawStan (iId := 1, bStan := FALSE);
	END_IF
//kontrola powrotu
	IF (tonCzasNaPowrot.Q) THEN
		fbLBKomunikacja.UstawStan (iId := 2, bStan := TRUE);
	ELSIF (fbCzujnikPozycja0.CzyZadzialany AND NOT bPrzesuwanieWStronePoczatku) THEN
		fbLBKomunikacja.UstawStan (iId := 2, bStan := FALSE);
	END_IF
//kontrola utraty pozycji 0
	fbKontrolaCzujnik0_F (CLK := fbCzujnikPozycja0.CzyZadzialany);
	IF (fbKontrolaCzujnik0_F.Q AND NOT bPrzesuwanieWStroneKonca) THEN
		fbLBKomunikacja.UstawStan (iId := 3, bStan := TRUE);
	ELSIF (fbCzujnikPozycja0.CzyZadzialany) THEN
		fbLBKomunikacja.UstawStan (iId := 3, bStan := FALSE);
	END_IF
//kontrola utraty pozycji MAX
	fbKontrolaCzujnikMax_F (CLK := fbCzujnikPozycjaMax.CzyZadzialany);
	IF (fbKontrolaCzujnikMax_F.Q AND NOT bPrzesuwanieWStronePoczatku) THEN
		fbLBKomunikacja.UstawStan (iId := 4, bStan := TRUE);
	ELSIF (fbCzujnikPozycjaMax.CzyZadzialany) THEN
		fbLBKomunikacja.UstawStan (iId := 4, bStan := FALSE);
	END_IF	
//Bladustawienia czujnikow - zadziałane dwa czujniki
	IF (fbCzujnikPozycja0.CzyZadzialany AND fbCzujnikPozycjaMax.CzyZadzialany) THEN
		fbLBKomunikacja.UstawStan (iId := 5, bStan := TRUE);
	ELSE
		fbLBKomunikacja.UstawStan (iId := 5, bStan := FALSE);
	END_IF
//Blad zamiany czujnikow	
	fbKontrolaCzujnik0_R (CLK := fbCzujnikPozycja0.CzyZadzialany);
	fbKontrolaCzujnikMax_R (CLK := fbCzujnikPozycjaMax.CzyZadzialany);
	IF ((fbKontrolaCzujnik0_R.Q AND bPrzesuwanieWStroneKonca) OR
		(fbKontrolaCzujnikMax_R.Q AND bPrzesuwanieWStronePoczatku)) THEN
		fbLBKomunikacja.UstawStan (iId := 6, bStan := FALSE);
	END_IF
	IF ((NaPoczatku AND NOT bPrzesuwanieWStroneKonca) OR 
		(NaKoncu and not bPrzesuwanieWStronePoczatku) ) THEN
		fbLBKomunikacja.UstawStan (iId := 6, bStan := FALSE);
	END_IF
END_METHOD

END_FUNCTION_BLOCK

// ---- POUs/01 - Elementy/Silownik/POU/FB_Silownik.TcPOU
//==================================================================================================
//								RJM Maszyny sp. z o.o.
//									13.05.2022
//	Obsługa silonwika podstawa
//	Realizacja wysuwania i chowania tłoczyska dla jednej cewki zwrócenie pozycji skrajnych
// 	v1.0	|| TC v 3.1.4024.22		|| - pierwsza wersja
//==================================================================================================
FUNCTION_BLOCK FB_Silownik IMPLEMENTS ITF_Silownik
VAR_INPUT
END_VAR
VAR_OUTPUT
END_VAR
VAR
	fbCzujnikPozycja0						: ITF_Czujnik;		//czujnik połozenia tłoczyska
	fbCzujnikPozycjaMax						: ITF_Czujnik;		//czujnik położenia tłoczyska
	fbElektrozawor							: ITF_Elektozawor;	//elektrozawor sterujący siłownikiem
	
	bPrzesuwanieWStronePoczatku				: BOOL;
	bPrzesuwanieWStroneKonca				: BOOL;
END_VAR

METHOD FB_init : BOOL
VAR_INPUT
	bInitRetains : BOOL; // if TRUE, the retain variables are initialized (warm start / cold start)
	bInCopyCode : BOOL;  // if TRUE, the instance afterwards gets moved into the copy code (online change)
	fbCzujnikPozycja0						: ITF_Czujnik;		//czujnik połozenia tłoczyska
	fbCzujnikPozycjaMax						: ITF_Czujnik;		//czujnik położenia tłoczyska
	fbElektrozawor							: ITF_Elektozawor;	//elektrozawor sterujący siłownikiem
END_VAR
THIS^.fbCzujnikPozycja0						:= fbCzujnikPozycja0;	  
THIS^.fbCzujnikPozycjaMax					:= fbCzujnikPozycjaMax;
THIS^.fbElektrozawor						:= fbElektrozawor;
END_METHOD

//==================================================================================================
//								RJM Maszyny sp. z o.o.
//									13.05.2022
//	Informacja tłoczysko na końcu
// 	v1.0	|| TC v 3.1.4024.22		|| - pierwsza wersja
//==================================================================================================
PROPERTY NaKoncu : BOOL
GET
IF (fbCzujnikPozycjaMax.CzyZadzialany AND NOT bPrzesuwanieWStroneKonca) THEN
	NaKoncu									:= TRUE;
ELSE
	NaKoncu									:= FALSE;
END_IF
END_GET
END_PROPERTY

//==================================================================================================
//								RJM Maszyny sp. z o.o.
//									13.05.2022
//	Informacja tłoczysko na początku
// 	v1.0	|| TC v 3.1.4024.22		|| - pierwsza wersja
//==================================================================================================
PROPERTY NaPoczatku : BOOL
GET
IF (fbCzujnikPozycja0.CzyZadzialany AND NOT bPrzesuwanieWStronePoczatku) THEN
	NaPoczatku								:= TRUE;
ELSE
	NaPoczatku								:= FALSE;
END_IF
END_GET
END_PROPERTY

//==================================================================================================
//								RJM Maszyny sp. z o.o.
//									13.05.2022
//	Metoda sterująca siłownikiem - MUSI BYĆ WYWOŁYWANA W KAŻDYM CYKLU PROGRAMU
// 	v1.0	|| TC v 3.1.4024.22		|| - pierwsza wersja
//==================================================================================================
METHOD Praca : BOOL
VAR_INPUT
END_VAR
//Flaga pomocnicza informacja o przesuwaniu w strone poczatku tłoczyska
IF (bPrzesuwanieWStronePoczatku AND fbCzujnikPozycja0.CzyZadzialany) THEN
	bPrzesuwanieWStronePoczatku				:= FALSE;
END_IF
//Flaga pomocnicza informacja o przesuwaniu w strone konca tłoczyska
IF (bPrzesuwanieWStroneKonca AND fbCzujnikPozycjaMax.CzyZadzialany) THEN
	bPrzesuwanieWStroneKonca				:= FALSE;
END_IF
END_METHOD

(*==================================================================================================
								RJM Maszyny sp. z o.o.
									13.05.2022
	Przesun tłoczysko w strone końca
 	v1.0	|| TC v 3.1.4024.22		|| - pierwsza wersja
==================================================================================================*)
PROPERTY PrzesunDoKonca : BOOL
SET
StanSilownika (bRuchWStronePoczatku	:= FALSE,
				bRuchWstroneKonca	:= TRUE);
END_SET
END_PROPERTY

(*==================================================================================================
								RJM Maszyny sp. z o.o.
									13.05.2022
	Przesun tłoczysko w strone poczatku
 	v1.0	|| TC v 3.1.4024.22		|| - pierwsza wersja
==================================================================================================*)
PROPERTY PrzesunDoPoczatku : BOOL
SET
StanSilownika (bRuchWStronePoczatku	:= TRUE,
				bRuchWstroneKonca	:= FALSE);
END_SET
END_PROPERTY

(*==================================================================================================
								RJM Maszyny sp. z o.o.
									13.05.2022
	Przesuwanie tłoczyska w strone końca
 	v1.0	|| TC v 3.1.4024.22		|| - pierwsza wersja
==================================================================================================*)
PROPERTY PrzesuwanieWStroneKonca : BOOL
GET
PrzesuwanieWStroneKonca						:= bprzesuwanieWStroneKonca;
END_GET
END_PROPERTY

(*==================================================================================================
								RJM Maszyny sp. z o.o.
									13.05.2022
	Przesuwanie tłoczyska w strone poczatku
 	v1.0	|| TC v 3.1.4024.22		|| - pierwsza wersja
==================================================================================================*)
PROPERTY PrzesuwanieWStronePoczatku : BOOL
GET
PrzesuwanieWStronePoczatku					:= bPrzesuwanieWStronePoczatku;
END_GET
END_PROPERTY

METHOD PROTECTED StanSilownika
VAR_INPUT
	bRuchWStronePoczatku					: BOOL;
	bRuchWstroneKonca						: BOOL;
END_VAR

IF (bRuchWStronePoczatku AND NOT bRuchWstroneKonca) THEN
	bPrzesuwanieWStronePoczatku				:= TRUE;
	bprzesuwanieWStroneKonca				:= FALSE;
	fbElektrozawor.Steruj (bKierunekWstrone0 := TRUE, bKierunekWStroneMax := FALSE);
END_IF
	

IF (bRuchWstroneKonca AND NOT bRuchWStronePoczatku) THEN
	bprzesuwanieWStroneKonca				:= TRUE;
	bPrzesuwanieWStronePoczatku				:= FALSE;
	fbElektrozawor.Steruj (bKierunekWstrone0 := FALSE, bKierunekWStroneMax := TRUE);
END_IF
END_METHOD

END_FUNCTION_BLOCK

// ---- POUs/01 - Elementy/Silownik/POU/FB_Silownik_Kontrola_Komunikacja.TcPOU
//==================================================================================================
//								RJM Maszyny sp. z o.o.
//									14.06.2022
//	FB posredniczący pomiędzy FB a logerem alarmów  
// 	v1.0	|| TC v 3.1.4024.22		|| - pierwsza wersja
//==================================================================================================
FUNCTION_BLOCK FB_Silownik_Kontrola_Komunikacja EXTENDS FB_LogowanieBledow_ElementWykonawczy
VAR_INPUT
END_VAR
VAR_OUTPUT
END_VAR
VAR
	
END_VAR

METHOD DefinicjaTabeliZdarzen_1031_Niemiecki : BOOL
VAR_INPUT
	arrTablicaDefinicjiZdarzenOpis			: REFERENCE TO ARRAY [1..GVL_LogowanieBledow_Stale.MAX_ILOSC_ZDARZEN] OF DUT_LogowanieBledow_ZdarzenieOpis;

END_VAR
arrTablicaDefinicjiZdarzenOpis [iStartId+0].sOpis	:= 'DE - zbyt dlugi czas w stronę końca';
arrTablicaDefinicjiZdarzenOpis [iStartId+1].sOpis	:= 'DE - zbyt dlugi czas w stronę początku';
arrTablicaDefinicjiZdarzenOpis [iStartId+2].sOpis	:= 'DE - utrata pozycji 0';
arrTablicaDefinicjiZdarzenOpis [iStartId+3].sOpis	:= 'DE - utrata pozycji MAX';
arrTablicaDefinicjiZdarzenOpis [iStartId+4].sOpis	:= 'DE - blad ustawienia czujnikow - dwa czujniki aktywne';
arrTablicaDefinicjiZdarzenOpis [iStartId+5].sOpis	:= 'DE - blad ustawiania ustawienia czujników - zamienione miejscami';
END_METHOD

METHOD DefinicjaTabeliZdarzen_1033_Angielski : BOOL
VAR_INPUT
	arrTablicaDefinicjiZdarzenOpis			: REFERENCE TO ARRAY [1..GVL_LogowanieBledow_Stale.MAX_ILOSC_ZDARZEN] OF DUT_LogowanieBledow_ZdarzenieOpis;

END_VAR
arrTablicaDefinicjiZdarzenOpis [iStartId+0].sOpis	:= 'EN - zbyt dlugi czas w stronę końca';
arrTablicaDefinicjiZdarzenOpis [iStartId+1].sOpis	:= 'EN - zbyt dlugi czas w stronę początku';
arrTablicaDefinicjiZdarzenOpis [iStartId+2].sOpis	:= 'EN - utrata pozycji 0';
arrTablicaDefinicjiZdarzenOpis [iStartId+3].sOpis	:= 'EN - utrata pozycji MAX';
arrTablicaDefinicjiZdarzenOpis [iStartId+4].sOpis	:= 'EN - blad ustawienia czujnikow - dwa czujniki aktywne';
arrTablicaDefinicjiZdarzenOpis [iStartId+5].sOpis	:= 'EN - blad ustawiania ustawienia czujników - zamienione miejscami';
END_METHOD

METHOD DefinicjaTabeliZdarzen_1045_Polski : BOOL
VAR_INPUT
	arrTablicaDefinicjiZdarzenOpis			: REFERENCE TO ARRAY [1..GVL_LogowanieBledow_Stale.MAX_ILOSC_ZDARZEN] OF DUT_LogowanieBledow_ZdarzenieOpis;

END_VAR
arrTablicaDefinicjiZdarzenOpis [iStartId+0].sOpis	:= 'PL - zbyt dlugi czas w stronę końca';
arrTablicaDefinicjiZdarzenOpis [iStartId+1].sOpis	:= 'PL - zbyt dlugi czas w stronę początku';
arrTablicaDefinicjiZdarzenOpis [iStartId+2].sOpis	:= 'PL - utrata pozycji 0';
arrTablicaDefinicjiZdarzenOpis [iStartId+3].sOpis	:= 'PL - utrata pozycji MAX';
arrTablicaDefinicjiZdarzenOpis [iStartId+4].sOpis	:= 'PL - blad ustawienia czujnikow - dwa czujniki aktywne';
arrTablicaDefinicjiZdarzenOpis [iStartId+5].sOpis	:= 'PL - blad ustawiania ustawienia czujników - zamienione miejscami';
END_METHOD

METHOD DefinicjaTabeliZdarzen_Ogolna : BOOL
VAR_INPUT
	arrTablicaDefinicjiZdarzen				: REFERENCE TO ARRAY [1..GVL_LogowanieBledow_Stale.MAX_ILOSC_ZDARZEN] OF DUT_LogowanieBledow_Zdarzenie;
	arrTablicaDefinicjiZdarzenOpis			: REFERENCE TO ARRAY [1..GVL_LogowanieBledow_Stale.MAX_ILOSC_ZDARZEN] OF DUT_LogowanieBledow_ZdarzenieOpis;
	arrTablicaDefinicjiZdarzenStan			: REFERENCE TO ARRAY [1..GVL_LogowanieBledow_Stale.MAX_ILOSC_ZDARZEN] OF DUT_LogowanieBledow_ZdarzenieStan;

	iIdZdarzenia							: REFERENCE TO INT;
	iNrPodzespolu							: INT := 0;
	iNrPodelementu							: INT := 0;
	iNrElementu								: INT := 0;
END_VAR
//zbyt dlugi czas w stronę końca
	iIdZdarzenia										:= iIdZdarzenia + 1;
	arrTablicaDefinicjiZdarzen [iIdZdarzenia].iIdZdarzenia			:= iIdZdarzenia;
	arrTablicaDefinicjiZdarzen [iIdZdarzenia].byRodzajZdarzenia	:= 2;
	arrTablicaDefinicjiZdarzen [iIdZdarzenia].sKodBledu			:= '0001';
	arrTablicaDefinicjiZdarzen [iIdZdarzenia].sNrKomponentu		:= GenerujNrKomponentu (iNrPodzespolu := iNrPodzespolu, iNrPodelementu := iNrPodelementu, iNrElementu := iNrElementu); 
	arrTablicaDefinicjiZdarzenOpis [iIdZdarzenia].iIdZdarzenia 	:= iIdZdarzenia;
	arrTablicaDefinicjiZdarzenStan [iIdZdarzenia].iIdZdarzenia 	:= iIdZdarzenia;
	arrTablicaDefinicjiZdarzenStan [iIdZdarzenia].bAktywne			:= FALSE;
//zbyt dlugi czas w stronę początku	
	iIdZdarzenia										:= iIdZdarzenia + 1;
	arrTablicaDefinicjiZdarzen [iIdZdarzenia].iIdZdarzenia			:= iIdZdarzenia;
	arrTablicaDefinicjiZdarzen [iIdZdarzenia].byRodzajZdarzenia	:= 2;
	arrTablicaDefinicjiZdarzen [iIdZdarzenia].sKodBledu			:= '0002';
	arrTablicaDefinicjiZdarzen [iIdZdarzenia].sNrKomponentu		:= GenerujNrKomponentu (iNrPodzespolu := iNrPodzespolu, iNrPodelementu := iNrPodelementu, iNrElementu := iNrElementu); 
	arrTablicaDefinicjiZdarzenOpis [iIdZdarzenia].iIdZdarzenia 	:= iIdZdarzenia;
	arrTablicaDefinicjiZdarzenStan [iIdZdarzenia].iIdZdarzenia 	:= iIdZdarzenia;
	arrTablicaDefinicjiZdarzenStan [iIdZdarzenia].bAktywne			:= FALSE;
//utrata pozycji 0
	iIdZdarzenia										:= iIdZdarzenia + 1;
	arrTablicaDefinicjiZdarzen [iIdZdarzenia].iIdZdarzenia			:= iIdZdarzenia;
	arrTablicaDefinicjiZdarzen [iIdZdarzenia].byRodzajZdarzenia	:= 2;
	arrTablicaDefinicjiZdarzen [iIdZdarzenia].sKodBledu			:= '0003';
	arrTablicaDefinicjiZdarzen [iIdZdarzenia].sNrKomponentu 		:= GenerujNrKomponentu (iNrPodzespolu := iNrPodzespolu, iNrPodelementu := iNrPodelementu, iNrElementu := iNrElementu); 
	arrTablicaDefinicjiZdarzenOpis [iIdZdarzenia].iIdZdarzenia 	:= iIdZdarzenia;
	arrTablicaDefinicjiZdarzenStan [iIdZdarzenia].iIdZdarzenia 	:= iIdZdarzenia;
	arrTablicaDefinicjiZdarzenStan [iIdZdarzenia].bAktywne			:= FALSE;
//utrata pozycji MAX
	iIdZdarzenia										:= iIdZdarzenia + 1;
	arrTablicaDefinicjiZdarzen [iIdZdarzenia].iIdZdarzenia			:= iIdZdarzenia;
	arrTablicaDefinicjiZdarzen [iIdZdarzenia].byRodzajZdarzenia	:= 2;
	arrTablicaDefinicjiZdarzen [iIdZdarzenia].sKodBledu			:= '0004';
	arrTablicaDefinicjiZdarzen [iIdZdarzenia].sNrKomponentu 		:= GenerujNrKomponentu (iNrPodzespolu := iNrPodzespolu, iNrPodelementu := iNrPodelementu, iNrElementu := iNrElementu); 
	arrTablicaDefinicjiZdarzenOpis [iIdZdarzenia].iIdZdarzenia 	:= iIdZdarzenia;
	arrTablicaDefinicjiZdarzenStan [iIdZdarzenia].iIdZdarzenia 	:= iIdZdarzenia;
	arrTablicaDefinicjiZdarzenStan [iIdZdarzenia].bAktywne			:= FALSE;
//blad ustawienia czujnikow - dwa czujniki aktywne
	iIdZdarzenia										:= iIdZdarzenia + 1;
	arrTablicaDefinicjiZdarzen [iIdZdarzenia].iIdZdarzenia			:= iIdZdarzenia;
	arrTablicaDefinicjiZdarzen [iIdZdarzenia].byRodzajZdarzenia	:= 1;
	arrTablicaDefinicjiZdarzen [iIdZdarzenia].sKodBledu			:= '0005';
	arrTablicaDefinicjiZdarzen [iIdZdarzenia].sNrKomponentu 		:= GenerujNrKomponentu (iNrPodzespolu := iNrPodzespolu, iNrPodelementu := iNrPodelementu, iNrElementu := iNrElementu); 
	arrTablicaDefinicjiZdarzenOpis [iIdZdarzenia].iIdZdarzenia 	:= iIdZdarzenia;
	arrTablicaDefinicjiZdarzenStan [iIdZdarzenia].iIdZdarzenia 	:= iIdZdarzenia;
	arrTablicaDefinicjiZdarzenStan [iIdZdarzenia].bAktywne			:= FALSE;
//blad ustawiania ustawienia czujników - zamienione miejscami	
	iIdZdarzenia										:= iIdZdarzenia + 1;
	arrTablicaDefinicjiZdarzen [iIdZdarzenia].iIdZdarzenia			:= iIdZdarzenia;
	arrTablicaDefinicjiZdarzen [iIdZdarzenia].byRodzajZdarzenia	:= 1;
	arrTablicaDefinicjiZdarzen [iIdZdarzenia].sKodBledu			:= '0006';
	arrTablicaDefinicjiZdarzen [iIdZdarzenia].sNrKomponentu 		:= GenerujNrKomponentu (iNrPodzespolu := iNrPodzespolu, iNrPodelementu := iNrPodelementu, iNrElementu := iNrElementu); 
	arrTablicaDefinicjiZdarzenOpis [iIdZdarzenia].iIdZdarzenia 	:= iIdZdarzenia;
	arrTablicaDefinicjiZdarzenStan [iIdZdarzenia].iIdZdarzenia 	:= iIdZdarzenia;
	arrTablicaDefinicjiZdarzenStan [iIdZdarzenia].bAktywne			:= FALSE;
END_METHOD

END_FUNCTION_BLOCK

// ---- POUs/95 - Logowanie bledow/POU/FB_LogowanieBledow_ElementWykonawczy.TcPOU
//==================================================================================================
//								RJM Maszyny sp. z o.o.
//									14.06.2022
//	FB posredniczący pomiędzy FB a logerem alarmów  
// 	v1.0	|| TC v 3.1.4024.22		|| - pierwsza wersja
//==================================================================================================
FUNCTION_BLOCK FB_LogowanieBledow_ElementWykonawczy IMPLEMENTS ITF_LogowanieBledow_ElementWykonawczy
VAR_INPUT
END_VAR
VAR_OUTPUT
END_VAR
VAR
	iStartId								: INT := 0;	//numer poczatkowy dla podzespolu
	arrTablicaStanow						: ARRAY [1..GVL_LogowanieBledow_Stale.MAX_ILOSC_ZDARZEN_NA_ELEMENT] OF BOOL;
END_VAR

//==================================================================================================
//								RJM Maszyny sp. z o.o.
//									14.06.2022
//	Metoda do rozszerzenia z opisem alarmów po niemiecku  
// 	v1.0	|| TC v 3.1.4024.22		|| - pierwsza wersja
//==================================================================================================
METHOD DefinicjaTabeliZdarzen_1031_Niemiecki : BOOL
VAR_INPUT
	arrTablicaDefinicjiZdarzenOpis			: REFERENCE TO ARRAY [1..GVL_LogowanieBledow_Stale.MAX_ILOSC_ZDARZEN] OF DUT_LogowanieBledow_ZdarzenieOpis;

END_VAR
END_METHOD

//==================================================================================================
//								RJM Maszyny sp. z o.o.
//									14.06.2022
//	Metoda do rozszerzenia z opisem alarmów po andgielsku  
// 	v1.0	|| TC v 3.1.4024.22		|| - pierwsza wersja
//==================================================================================================
METHOD DefinicjaTabeliZdarzen_1033_Angielski : BOOL
VAR_INPUT
	arrTablicaDefinicjiZdarzenOpis			: REFERENCE TO ARRAY [1..GVL_LogowanieBledow_Stale.MAX_ILOSC_ZDARZEN] OF DUT_LogowanieBledow_ZdarzenieOpis;

END_VAR
END_METHOD

//==================================================================================================
//								RJM Maszyny sp. z o.o.
//									14.06.2022
//	Metoda do rozszerzenia z opisem alarmów po polsku
// 	v1.0	|| TC v 3.1.4024.22		|| - pierwsza wersja
//==================================================================================================
METHOD DefinicjaTabeliZdarzen_1045_Polski : BOOL
VAR_INPUT
	arrTablicaDefinicjiZdarzenOpis			: REFERENCE TO ARRAY [1..GVL_LogowanieBledow_Stale.MAX_ILOSC_ZDARZEN] OF DUT_LogowanieBledow_ZdarzenieOpis;

END_VAR
END_METHOD

//==================================================================================================
//								RJM Maszyny sp. z o.o.
//									14.06.2022
//	Metoda do rozszerzenia wypełniająca niezmienne dane tablic  
// 	v1.0	|| TC v 3.1.4024.22		|| - pierwsza wersja
//==================================================================================================
METHOD DefinicjaTabeliZdarzen_Ogolna : BOOL
VAR_INPUT
	arrTablicaDefinicjiZdarzen				: REFERENCE TO ARRAY [1..GVL_LogowanieBledow_Stale.MAX_ILOSC_ZDARZEN] OF DUT_LogowanieBledow_Zdarzenie;
	arrTablicaDefinicjiZdarzenOpis			: REFERENCE TO ARRAY [1..GVL_LogowanieBledow_Stale.MAX_ILOSC_ZDARZEN] OF DUT_LogowanieBledow_ZdarzenieOpis;
	arrTablicaDefinicjiZdarzenStan			: REFERENCE TO ARRAY [1..GVL_LogowanieBledow_Stale.MAX_ILOSC_ZDARZEN] OF DUT_LogowanieBledow_ZdarzenieStan;

	iIdZdarzenia							: REFERENCE TO INT;
	iNrPodzespolu							: INT := 0;
	iNrPodelementu							: INT := 0;
	iNrElementu								: INT := 0;
END_VAR
END_METHOD

//==================================================================================================
//								RJM Maszyny sp. z o.o.
//									14.06.2022
//	Metoda składa numer podzespołu z podanych zmiennych 
// 	v1.0	|| TC v 3.1.4024.22		|| - pierwsza wersja
//==================================================================================================
METHOD GenerujNrKomponentu : STRING
VAR_INPUT
	iNrPodzespolu							: INT := 0;
	iNrPodelementu							: INT := 0;
	iNrElementu								: INT := 0;
END_VAR
VAR
	sKod									: STRING;
END_VAR
sKod										:= concat (TO_STRING (iNrPodzespolu*100), '-');
sKod										:= concat (sKod, TO_STRING (iNrPodelementu*10));
sKod										:= concat (sKod, '-');
sKod										:= concat (sKod, TO_STRING (iNrElementu));

GenerujNrKomponentu							:= sKod;
END_METHOD

//==================================================================================================
//								RJM Maszyny sp. z o.o.
//									14.06.2022
//	Przypisanie odpowiedniego stonu w odpowienim miejscu w tabeli potrzebne do aktualizacji stanow alarmow
// 	v1.0	|| TC v 3.1.4024.22		|| - pierwsza wersja
//==================================================================================================
METHOD UstawStan : BOOL
VAR_INPUT
	iId										: INT;
	bStan									: BOOL;
END_VAR
arrTablicaStanow [iId]					:= bStan;
END_METHOD

//==================================================================================================
//								RJM Maszyny sp. z o.o.
//									14.06.2022
//	Metoda zwraca definicje alarmow dla elementów wykonawczych
// 	v1.0	|| TC v 3.1.4024.22		|| - pierwsza wersja
//==================================================================================================
METHOD ZwrocTabliceDefinicji : BOOL
VAR_INPUT
	arrTablicaDefinicjiZdarzen				: REFERENCE TO ARRAY [1..GVL_LogowanieBledow_Stale.MAX_ILOSC_ZDARZEN] OF DUT_LogowanieBledow_Zdarzenie;
	arrTablicaDefinicjiZdarzenOpis			: REFERENCE TO ARRAY [1..GVL_LogowanieBledow_Stale.MAX_ILOSC_ZDARZEN] OF DUT_LogowanieBledow_ZdarzenieOpis;
	arrTablicaDefinicjiZdarzenStan			: REFERENCE TO ARRAY [1..GVL_LogowanieBledow_Stale.MAX_ILOSC_ZDARZEN] OF DUT_LogowanieBledow_ZdarzenieStan;
	
	iIdZdarzenia							: REFERENCE TO INT;
	iNrPodzespolu							: INT;
	iNrPodelementu							: INT;
	iNrElementu								: INT;
	iJezykId								: INT;
END_VAR
	IF (iStartId = 0) THEN
		iStartId							:= iIdZdarzenia+1;
		DefinicjaTabeliZdarzen_Ogolna (	arrTablicaDefinicjiZdarzen 		:= arrTablicaDefinicjiZdarzen,
										arrTablicaDefinicjiZdarzenOpis 	:= arrTablicaDefinicjiZdarzenOpis,
										arrTablicaDefinicjiZdarzenStan 	:= arrTablicaDefinicjiZdarzenStan,
										iIdZdarzenia 					:= iIdZdarzenia,
										iNrPodzespolu 					:= iNrPodzespolu,
										iNrPodelementu 					:= iNrPodelementu,
										iNrElementu						:= iNrElementu);
	END_IF
	
	CASE iJezykId OF
		1031	:	//niemiecki
			DefinicjaTabeliZdarzen_1031_Niemiecki (arrTablicaDefinicjiZdarzenOpis 	:= arrTablicaDefinicjiZdarzenOpis);
		1033	:	//angielski
			DefinicjaTabeliZdarzen_1033_Angielski (arrTablicaDefinicjiZdarzenOpis 	:= arrTablicaDefinicjiZdarzenOpis);
		1045	:	//polski
			DefinicjaTabeliZdarzen_1045_Polski (arrTablicaDefinicjiZdarzenOpis 	:= arrTablicaDefinicjiZdarzenOpis);
		ELSE		//domyslny polski
			DefinicjaTabeliZdarzen_1045_Polski (arrTablicaDefinicjiZdarzenOpis 	:= arrTablicaDefinicjiZdarzenOpis);		
	END_CASE
	
//	ZwrocTabeleZdarzen						REF= arrZdarzeniaDefinicja;
END_METHOD

//==================================================================================================
//								RJM Maszyny sp. z o.o.
//									14.06.2022
//	Metoda zwraca tablice stanow elementu wykonwaczego  
// 	v1.0	|| TC v 3.1.4024.22		|| - pierwsza wersja
//==================================================================================================
METHOD ZwrocTabliceStanu : BOOL
VAR_INPUT
	arrTablicaDefinicjiZdarzenStan			: REFERENCE TO ARRAY [1..GVL_LogowanieBledow_Stale.MAX_ILOSC_ZDARZEN] OF DUT_LogowanieBledow_ZdarzenieStan;
END_VAR

VAR
	iI: INT;
END_VAR
FOR iI := 1 TO 10 DO
	arrTablicaDefinicjiZdarzenStan [iStartId + iI -1].bAktywne := arrTablicaStanow [iI];
END_FOR
END_METHOD

END_FUNCTION_BLOCK

// ---- POUs/80 - Symulacja pracy/POU/FB_Symulacja.TcPOU
FUNCTION_BLOCK FB_Symulacja IMPLEMENTS ITF_StanMaszyny
VAR_INPUT
	stParametry								: DUT_Symulacja_Parametry;
	stStanyPodzespolow						: DUT_Krajalnica_StanyPodzespolow;
	eTrybPracy								: E_PMLUnitMode;
END_VAR
VAR_OUTPUT
	//wyjscia zadziałania czujnikow 
	bCiecie1_Poczatek						: BOOL;
	bCiecie1_Koniec							: BOOL;
	bCiecie2_Poczatek						: BOOL;
	bCiecie2_Koniec							: BOOL;
	bPodawanieZabierakPoczatek				: BOOL;
	bPodawanieZabierakKoniec				: BOOL;
	bPodawaniePrzesuwaniePoczatek			: BOOL;
	bPodawaniePrzesuwanieKoniec				: BOOL;
	bCzujnikWaflaDoPodania					: BOOL;
	bCzujnikWaflaDoCiecia1					: BOOL;
	bCzujnikWaflaDoCiecia2					: BOOL;
END_VAR
VAR
	tonCiecie1_BazowanieCzasNaPowrot				: TON;           
	tonCiecie1_CiecieCzasNaCiecie					: TON;
	tonCiecie1_CiecieCzasNaPowrot					: TON;
	tonCiecie2_BazowanieCzasNaPowrot				: TON;
	tonCiecie2_CiecieCzasNaCiecie					: TON;
	tonCiecie2_CiecieCzasNaPowrot					: TON;
	tonPodawanieZabierak_BazowanieCzasNaPowrot		: TON;
	tonPodawaniePrzesuwanie_BazowanieCzasNaPowrot	: TON;
	tonPodawanieZabierak_PodawanieCzasNaPrace	: TON;
	tonPodawanieZabierak_PodawanieCzasNaPowrot		: TON;
	tonPodawaniePrzesuwanie_PodawanieCzasNaPobranie	: TON;
	tonPodawaniePrzesuwanie_PodawanieCzasNaPodanie	: TON;	
END_VAR

tonCiecie1_BazowanieCzasNaPowrot				(IN := stStanyPodzespolow.bCiecie1_Bazowanie ,
													PT := REAL_TO_TIME (stParametry.rCiecie1_BazowanieCzasNaPowrot));
tonCiecie1_CiecieCzasNaCiecie					(IN := stStanyPodzespolow.bCiecie1_Naped_WStroneKonca ,
													PT := REAL_TO_TIME (stParametry.rCiecie1_CiecieCzasNaPowrot));
tonCiecie1_CiecieCzasNaPowrot					(IN := stStanyPodzespolow.bCiecie1_Naped_WStronePoczatku ,
													PT := REAL_TO_TIME (stParametry.rCiecie1_CiecieCzasNaCiecie));

tonCiecie2_BazowanieCzasNaPowrot				(IN := stStanyPodzespolow.bCiecie2_Bazowanie ,
													PT := REAL_TO_TIME (stParametry.rCiecie2_BazowanieCzasNaPowrot));
tonCiecie2_CiecieCzasNaCiecie					(IN := stStanyPodzespolow.bCiecie2_Naped_WStroneKonca ,
													PT := REAL_TO_TIME (stParametry.rCiecie2_CiecieCzasNaPowrot));
tonCiecie2_CiecieCzasNaPowrot					(IN := stStanyPodzespolow.bCiecie2_Naped_WStronePoczatku ,
													PT := REAL_TO_TIME (stParametry.rCiecie2_CiecieCzasNaCiecie));

tonPodawanieZabierak_BazowanieCzasNaPowrot		(IN := stStanyPodzespolow.bPodawanie_Bazowanie AND 
														stStanyPodzespolow.bPodawanie_Zabierak_WStronePoczatku ,
													PT := REAL_TO_TIME (stParametry.rPodawanieZabierak_BazowanieCzasNaPowrot));
tonPodawaniePrzesuwanie_BazowanieCzasNaPowrot	(IN := stStanyPodzespolow.bPodawanie_Bazowanie AND 
														stStanyPodzespolow.bPodawanie_Przesuwanie_WStronePoczatku ,
													PT := REAL_TO_TIME (stParametry.rPodawanieZabierak_PodawanieCzasNaPowrot));
tonPodawanieZabierak_PodawanieCzasNaPrace		(IN := stStanyPodzespolow.bPodawanie_Podawanie AND
														stStanyPodzespolow.bPodawanie_zabierak_WStroneKonca ,
													PT := REAL_TO_TIME (stParametry.rPodawanieZabierak_PodawanieCzasNaPrace));
tonPodawanieZabierak_PodawanieCzasNaPowrot		(IN := stStanyPodzespolow.bPodawanie_Podawanie AND
														stStanyPodzespolow.bPodawanie_Zabierak_WStronePoczatku ,
													PT := REAL_TO_TIME (stParametry.rPodawaniePrzesuwanie_BazowanieCzasNaPowrot));
tonPodawaniePrzesuwanie_PodawanieCzasNaPobranie	(IN := stStanyPodzespolow.bPodawanie_Podawanie AND
														stStanyPodzespolow.bPodawanie_Przesuwanie_WStroneKonca ,
													PT := REAL_TO_TIME (stParametry.rPodawaniePrzesuwanie_PodawanieCzasNaPobranie));
tonPodawaniePrzesuwanie_PodawanieCzasNaPodanie	(IN := stStanyPodzespolow.bPodawanie_Podawanie AND
														stStanyPodzespolow.bPodawanie_Przesuwanie_WStronePoczatku ,
													PT := REAL_TO_TIME (stParametry.rPodawaniePrzesuwanie_PodawanieCzasNaPodanie));

(*==================================================================================================
								RJM Maszyny sp. z o.o.
									5.06.2022
	Stan maszyny Aborted - metoda pusta
 	v1.0	|| TC v 3.1.4024.29		|| - pierwsza wersja
==================================================================================================*)
METHOD SM_Aborted : BOOL
END_METHOD

(*==================================================================================================
								RJM Maszyny sp. z o.o.
									5.06.2022
	Stan maszyny Aborting - awaryjne zatrzymanie maszyny E-STOP
 	v1.0	|| TC v 3.1.4024.29		|| - pierwsza wersja
==================================================================================================*)
METHOD SM_Aborting : BOOL
SM_Aborting									:= TRUE;
END_METHOD

(*==================================================================================================
								RJM Maszyny sp. z o.o.
									5.06.2022
	Stan maszyny Clearing
 	v1.0	|| TC v 3.1.4024.29		|| - pierwsza wersja
==================================================================================================*)
METHOD SM_Clearing : BOOL
SM_Clearing									:= TRUE;
END_METHOD

(*==================================================================================================
								RJM Maszyny sp. z o.o.
									5.06.2022
	Stan maszyny Complete 
 	v1.0	|| TC v 3.1.4024.29		|| - pierwsza wersja
==================================================================================================*)
METHOD SM_Complete : BOOL
END_METHOD

(*==================================================================================================
								RJM Maszyny sp. z o.o.
									5.06.2022
	Stan maszyny Completing
 	v1.0	|| TC v 3.1.4024.29		|| - pierwsza wersja
==================================================================================================*)
METHOD SM_Completing : BOOL
END_METHOD

(*==================================================================================================
								RJM Maszyny sp. z o.o.
									5.06.2022
	Stan maszyny Execute
 	v1.0	|| TC v 3.1.4024.29		|| - pierwsza wersja
==================================================================================================*)
METHOD SM_Execute : BOOL
VAR_INPUT
	eTrybPracy	: E_PMLUnitMode;
END_VAR
END_METHOD

(*==================================================================================================
								RJM Maszyny sp. z o.o.
									5.06.2022
	Stan maszyny Held  - metoda pusta
 	v1.0	|| TC v 3.1.4024.29		|| - pierwsza wersja
==================================================================================================*)
METHOD SM_Held : BOOL
END_METHOD

(*==================================================================================================
								RJM Maszyny sp. z o.o.
									5.06.2022
	Stan maszyny Holding
 	v1.0	|| TC v 3.1.4024.29		|| - pierwsza wersja
==================================================================================================*)
METHOD SM_Holding : BOOL
END_METHOD

(*==================================================================================================
								RJM Maszyny sp. z o.o.
									5.06.2022
	Stan maszyny Idle
 	v1.0	|| TC v 3.1.4024.29		|| - pierwsza wersja
==================================================================================================*)
METHOD SM_Idle : BOOL
END_METHOD

(*==================================================================================================
								RJM Maszyny sp. z o.o.
									5.06.2022
	Stan maszyny Reseting - konczenie niedokocznonych cykli i powrot podzespolami do pozycji startowej
 	v1.0	|| TC v 3.1.4024.29		|| - pierwsza wersja
==================================================================================================*)
METHOD SM_Resetting : BOOL
VAR_INPUT
	eTrybPracy								: E_PMLUnitMode;
END_VAR
SM_Resetting								:= TRUE;
END_METHOD

(*==================================================================================================
								RJM Maszyny sp. z o.o.
									5.06.2022
	Stan maszyny Starting - Ustawienie elementów do pracy 
 	v1.0	|| TC v 3.1.4024.29		|| - pierwsza wersja
==================================================================================================*)
METHOD SM_Starting : BOOL
END_METHOD

(*==================================================================================================
								RJM Maszyny sp. z o.o.
									5.06.2022
	Stan maszyny Stoped - metoda pusta
 	v1.0	|| TC v 3.1.4024.29		|| - pierwsza wersja
==================================================================================================*)
METHOD SM_Stopped : BOOL
END_METHOD

(*==================================================================================================
								RJM Maszyny sp. z o.o.
									5.06.2022
	Stan maszyny Stopping - Zakonczenie aktualnych operacji nie zaczynamy kolejnych
 	v1.0	|| TC v 3.1.4024.29		|| - pierwsza wersja
==================================================================================================*)
METHOD SM_Stopping : BOOL
END_METHOD

(*==================================================================================================
								RJM Maszyny sp. z o.o.
									5.06.2022
	Stan maszyny Suspended - metoda pusta
 	v1.0	|| TC v 3.1.4024.29		|| - pierwsza wersja
==================================================================================================*)
METHOD SM_Suspended : BOOL
END_METHOD

(*==================================================================================================
								RJM Maszyny sp. z o.o.
									5.06.2022
	Stan maszyny Suspending
 	v1.0	|| TC v 3.1.4024.29		|| - pierwsza wersja
==================================================================================================*)
METHOD SM_Suspending : BOOL
END_METHOD

(*==================================================================================================
								RJM Maszyny sp. z o.o.
									5.06.2022
	Stan maszyny Unholding
 	v1.0	|| TC v 3.1.4024.29		|| - pierwsza wersja
==================================================================================================*)
METHOD SM_Unholding : BOOL
END_METHOD

(*==================================================================================================
								RJM Maszyny sp. z o.o.
									5.06.2022
	Stan maszyny Unsuspending
 	v1.0	|| TC v 3.1.4024.29		|| - pierwsza wersja
==================================================================================================*)
METHOD SM_Unsuspending : BOOL
END_METHOD

END_FUNCTION_BLOCK

// ---- POUs/51 - Krajalnica/POU/FB_Krajalnica.TcPOU
//==================================================================================================
//								RJM Maszyny sp. z o.o.
//									5.06.2022
//	Sterowanie krajalnica  
// 	v1.0	|| TC v 3.1.4024.29		|| - pierwsza wersja
//==================================================================================================

FUNCTION_BLOCK FB_Krajalnica IMPLEMENTS ITF_StanMaszyny
VAR_INPUT
	stParametry								: DUT_Krajalnica_Parametry;
	stSterowanieSymulacja					: DUT_Krajalnica_Symulacja;
END_VAR
VAR_OUTPUT
	stStanyPodzespolow						: DUT_Krajalnica_StanyPodzespolow;
END_VAR
VAR
	bC1_Czujnik0							: ITF_Czujnik;
	bC1_CzujnikMax							: ITF_Czujnik;
	fbC1_Elektrozawor						: ITF_Elektozawor;
	bC2_Czujnik0							: ITF_Czujnik;
	bC2_CzujnikMax							: ITF_Czujnik;
	fbC2_Elektrozawor						: ITF_Elektozawor;
	bPW_Z_Czujnik0							: ITF_Czujnik;
	bPW_Z_CzujnikMax						: ITF_Czujnik;
	fbPW_Z_Elektrozawor						: ITF_Elektozawor;
	bPW_P_Czujnik0							: ITF_Czujnik;
	bPW_P_CzujnikMax						: ITF_Czujnik;
	fbPW_P_Elektrozawor						: ITF_Elektozawor;	
	bWafalNaWejsciu							: ITF_Czujnik;
	bWafalDoCiecia1							: ITF_Czujnik;
	bWafalDoCiecia2							: ITF_Czujnik;
	
	
	fbCiecie1								: FB_Ciecie (					bCzujnik0Naped			 	:= bC1_Czujnik0,
                                                            				bCzujnikMaxNaped		 	:= bC1_CzujnikMax,
                                                            				fbElektrozaworNaped		 	:= fbC1_Elektrozawor);
	fbCiecie2								: FB_Ciecie (					bCzujnik0Naped			 	:= bC2_Czujnik0,
                                                            				bCzujnikMaxNaped		 	:= bC2_CzujnikMax,
                                                            				fbElektrozaworNaped		 	:= fbC2_Elektrozawor);
	fbPodawanieWafla						: FB_PrzesuwaczNaSilowniku (	bCzujnik0Zabieraka			:= bPW_Z_Czujnik0,
                                                                            bCzujnikMaxZabieraka		:= bPW_Z_CzujnikMax,
                                                                            fbElektrozaworZabieraka		:= fbPW_Z_Elektrozawor,
                                                                            bCzujnik0Przesuwacza		:= bPW_P_Czujnik0,
                                                                            bCzujnikMaxPrzesuwacza		:= bPW_P_CzujnikMax,
                                                                            fbElektrozaworPrzesuwacza	:= fbPW_P_Elektrozawor);
	
	arrElementyWykonawcze 					: ARRAY [1..GVL_LogowanieBledow_Stale.MAX_ILOSC_ELEMENTOW_NA_PODZESPOL] OF ITF_LogowanieBledow_ElementWykonawczy := 
														[	fbCiecie1.fbLBKomunikacja,
															fbCiecie2.fbLBKomunikacja,
															fbPodawanieWafla.fbLBKomunikacja];
															
	fbLBKomunikacja							: FB_PrzesuwaczNaSilowniku_Komunikacja 
														(	arrElementyWykonawcze := arrElementyWykonawcze,
															iIloscPodlementow := 3);	
															
	bSM_Resetting_PierwszePrzejscie			: BOOL := FALSE;
														

END_VAR

fbCiecie1.Praca ();
fbCiecie2.Praca ();
fbPodawanieWafla.Praca ();

StanyPodzespolow ();

METHOD FB_init : BOOL
VAR_INPUT
	bInitRetains : BOOL; // if TRUE, the retain variables are initialized (warm start / cold start)
	bInCopyCode : BOOL;  // if TRUE, the instance afterwards gets moved into the copy code (online change)
	bC1_Czujnik0							: ITF_Czujnik;
	bC1_CzujnikMax							: ITF_Czujnik;
	fbC1_Elektrozawor						: ITF_Elektozawor;
	bC2_Czujnik0							: ITF_Czujnik;
	bC2_CzujnikMax							: ITF_Czujnik;
	fbC2_Elektrozawor						: ITF_Elektozawor;
	bPW_Z_Czujnik0							: ITF_Czujnik;
	bPW_Z_CzujnikMax						: ITF_Czujnik;
	fbPW_Z_Elektrozawor						: ITF_Elektozawor;
	bPW_P_Czujnik0							: ITF_Czujnik;
	bPW_P_CzujnikMax						: ITF_Czujnik;
	fbPW_P_Elektrozawor						: ITF_Elektozawor;
	bWafalNaWejsciu							: ITF_Czujnik;
	bWafalDoCiecia1							: ITF_Czujnik;
	bWafalDoCiecia2							: ITF_Czujnik;
END_VAR
THIS^.bC1_Czujnik0							:= bC1_Czujnik0;
THIS^.bC1_CzujnikMax						:= bC1_CzujnikMax;
THIS^.fbC1_Elektrozawor						:= fbC1_Elektrozawor;
THIS^.bC2_Czujnik0							:= bC2_Czujnik0;
THIS^.bC2_CzujnikMax						:= bC2_CzujnikMax;
THIS^.fbC2_Elektrozawor						:= fbC2_Elektrozawor;
THIS^.bPW_Z_Czujnik0						:= bPW_Z_Czujnik0; 
THIS^.bPW_Z_CzujnikMax						:= bPW_Z_CzujnikMax; 
THIS^.fbPW_Z_Elektrozawor					:= fbPW_Z_Elektrozawor; 
THIS^.bPW_P_Czujnik0						:= bPW_P_Czujnik0; 
THIS^.bPW_P_CzujnikMax						:= bPW_P_CzujnikMax; 
THIS^.fbPW_P_Elektrozawor					:= fbPW_P_Elektrozawor; 
THIS^.bWafalNaWejsciu						:= bWafalNaWejsciu;
THIS^.bWafalDoCiecia1						:= bWafalDoCiecia1;
THIS^.bWafalDoCiecia2						:= bWafalDoCiecia2;

THIS^.fbCiecie1.FB_init (FALSE, FALSE, bC1_Czujnik0, bC1_CzujnikMax, fbC1_Elektrozawor);	
THIS^.fbCiecie2.FB_init (FALSE, FALSE, bC2_Czujnik0, bC2_CzujnikMax, fbC2_Elektrozawor);
THIS^.fbPodawanieWafla.FB_init (FALSE, FALSE, bPW_Z_Czujnik0, bPW_Z_CzujnikMax, fbPW_Z_Elektrozawor, bPW_P_Czujnik0, bPW_P_CzujnikMax ,fbPW_P_Elektrozawor);
END_METHOD

//==================================================================================================
//								RJM Maszyny sp. z o.o.
//									5.06.2022
//	Stan maszyny Aborted - metoda pusta
// 	v1.0	|| TC v 3.1.4024.29		|| - pierwsza wersja
//==================================================================================================
METHOD SM_Aborted : BOOL
VAR_INPUT

END_VAR
END_METHOD

//==================================================================================================
//								RJM Maszyny sp. z o.o.
//									5.06.2022
//	Stan maszyny Aborting - awaryjne zatrzymanie maszyny E-STOP
// 	v1.0	|| TC v 3.1.4024.29		|| - pierwsza wersja
//==================================================================================================
METHOD SM_Aborting : BOOL
END_METHOD

//==================================================================================================
//								RJM Maszyny sp. z o.o.
//									5.06.2022
//	Stan maszyny Clearing
// 	v1.0	|| TC v 3.1.4024.29		|| - pierwsza wersja
//==================================================================================================
METHOD SM_Clearing : BOOL
SM_Clearing := TRUE;
END_METHOD

//==================================================================================================
//								RJM Maszyny sp. z o.o.
//									5.06.2022
//	Stan maszyny Complete 
// 	v1.0	|| TC v 3.1.4024.29		|| - pierwsza wersja
//==================================================================================================
METHOD SM_Complete : BOOL
END_METHOD

//==================================================================================================
//								RJM Maszyny sp. z o.o.
//									5.06.2022
//	Stan maszyny Completing
// 	v1.0	|| TC v 3.1.4024.29		|| - pierwsza wersja
//==================================================================================================
METHOD SM_Completing : BOOL
END_METHOD

//==================================================================================================
//								RJM Maszyny sp. z o.o.
//									5.06.2022
//	Stan maszyny Execute
// 	v1.0	|| TC v 3.1.4024.29		|| - pierwsza wersja
//==================================================================================================
METHOD SM_Execute : BOOL
VAR_INPUT
	eTrybPracy								: E_PMLUnitMode;
END_VAR
CASE eTrybPracy OF
	E_PMLUnitMode.MANUAL		:
		SM_Execute_Manual ();
	E_PMLUnitMode.SEMIAUTOMATIC	:
		SM_Execute_Semiautomatic ();
	E_PMLUnitMode.AUTOMATIC		:
		SM_Execute_Automatic ();
END_CASE
END_METHOD

METHOD PRIVATE SM_Execute_Automatic : BOOL
VAR_INPUT
END_VAR
END_METHOD

METHOD PRIVATE SM_Execute_Manual : BOOL
VAR_INPUT
END_VAR
END_METHOD

METHOD PRIVATE SM_Execute_Semiautomatic : BOOL
VAR_INPUT
END_VAR
END_METHOD

//==================================================================================================
//								RJM Maszyny sp. z o.o.
//									5.06.2022
//	Stan maszyny Held  - metoda pusta
// 	v1.0	|| TC v 3.1.4024.29		|| - pierwsza wersja
//==================================================================================================
METHOD SM_Held : BOOL
END_METHOD

//==================================================================================================
//								RJM Maszyny sp. z o.o.
//									5.06.2022
//	Stan maszyny Holding
// 	v1.0	|| TC v 3.1.4024.29		|| - pierwsza wersja
//==================================================================================================
METHOD SM_Holding : BOOL
END_METHOD

//==================================================================================================
//								RJM Maszyny sp. z o.o.
//									5.06.2022
//	Stan maszyny Idle
// 	v1.0	|| TC v 3.1.4024.29		|| - pierwsza wersja
//==================================================================================================
METHOD SM_Idle : BOOL
END_METHOD

//==================================================================================================
//								RJM Maszyny sp. z o.o.
//									5.06.2022
//	Stan maszyny Reseting - konczenie niedokocznonych cykli i powrot podzespolami do pozycji startowej
// 	v1.0	|| TC v 3.1.4024.29		|| - pierwsza wersja
//==================================================================================================
METHOD SM_Resetting : BOOL
VAR_INPUT
	eTrybPracy								: E_PMLUnitMode;
END_VAR

CASE eTrybPracy OF
	E_PMLUnitMode.MANUAL		:
		;
	E_PMLUnitMode.SEMIAUTOMATIC	:
		IF (stSterowanieSymulacja.bCiecie1Bazuj) THEN
			fbCiecie1.Bazuj							:= TRUE;
		END_IF
		IF (stSterowanieSymulacja.bCiecie1Tnij) THEN
			fbCiecie1.WykonajCyklPracy				:= TRUE;
		END_IF
		IF (stSterowanieSymulacja.bCiecie2Bazuj) THEN
			fbCiecie2.Bazuj							:= TRUE;
		END_IF
		IF (stSterowanieSymulacja.bCiecie2Tnij) THEN
			fbCiecie2.WykonajCyklPracy				:= TRUE;
		END_IF
		IF (stSterowanieSymulacja.bPodawanieBazuj) THEN
			fbPodawanieWafla.Bazuj					:= TRUE;
		END_IF
		IF (stSterowanieSymulacja.bPodawaniePodaj) THEN
			fbPodawanieWafla.WykonajCyklPracy		:= TRUE;
		END_IF
	E_PMLUnitMode.AUTOMATIC		:
		(*
		DOPISAĆ KOŃCZENIE CYKLI JAK ZOSTAŁY PRZERWANE
		*)
		IF (NOT bSM_Resetting_PierwszePrzejscie) THEN
			fbCiecie1.Bazuj							:= TRUE;
			fbCiecie2.Bazuj							:= TRUE;
			fbPodawanieWafla.Bazuj					:= TRUE;
			bSM_Resetting_PierwszePrzejscie			:= TRUE;
		END_IF
		
		IF (fbCiecie1.Pozycja0 AND fbCiecie2.Pozycja0 AND fbPodawanieWafla.Pozycja0) THEN
			SM_Resetting 							:= TRUE;
			bSM_Resetting_PierwszePrzejscie			:= FALSE;
		ELSE
			SM_Resetting							:= FALSE;
		END_IF
END_CASE
END_METHOD

//==================================================================================================
//								RJM Maszyny sp. z o.o.
//									5.06.2022
//	Stan maszyny Starting - Ustawienie elementów do pracy 
// 	v1.0	|| TC v 3.1.4024.29		|| - pierwsza wersja
//==================================================================================================
METHOD SM_Starting : BOOL
SM_Starting 								:= TRUE;
END_METHOD

//==================================================================================================
//								RJM Maszyny sp. z o.o.
//									5.06.2022
//	Stan maszyny Stoped - metoda pusta
// 	v1.0	|| TC v 3.1.4024.29		|| - pierwsza wersja
//==================================================================================================
METHOD SM_Stopped : BOOL
END_METHOD

//==================================================================================================
//								RJM Maszyny sp. z o.o.
//									5.06.2022
//	Stan maszyny Stopping - Zakonczenie aktualnych operacji nie zaczynamy kolejnych
// 	v1.0	|| TC v 3.1.4024.29		|| - pierwsza wersja
//==================================================================================================
METHOD SM_Stopping : BOOL
END_METHOD

//==================================================================================================
//								RJM Maszyny sp. z o.o.
//									5.06.2022
//	Stan maszyny Suspended - metoda pusta
// 	v1.0	|| TC v 3.1.4024.29		|| - pierwsza wersja
//==================================================================================================
METHOD SM_Suspended : BOOL
END_METHOD

//==================================================================================================
//								RJM Maszyny sp. z o.o.
//									5.06.2022
//	Stan maszyny Suspending
// 	v1.0	|| TC v 3.1.4024.29		|| - pierwsza wersja
//==================================================================================================
METHOD SM_Suspending : BOOL
END_METHOD

//==================================================================================================
//								RJM Maszyny sp. z o.o.
//									5.06.2022
//	Stan maszyny Unholding
// 	v1.0	|| TC v 3.1.4024.29		|| - pierwsza wersja
//==================================================================================================
METHOD SM_Unholding : BOOL
END_METHOD

//==================================================================================================
//								RJM Maszyny sp. z o.o.
//									5.06.2022
//	Stan maszyny Unsuspending
// 	v1.0	|| TC v 3.1.4024.29		|| - pierwsza wersja
//==================================================================================================
METHOD SM_Unsuspending : BOOL
END_METHOD

METHOD StanyPodzespolow : DUT_Krajalnica_StanyPodzespolow
VAR_INPUT
END_VAR
stStanyPodzespolow.bCiecie1_Bazowanie						:= fbCiecie1.Bazowanie;
stStanyPodzespolow.bCiecie1_Ciecie							:= fbCiecie1.CyklPracy;
stStanyPodzespolow.bCiecie1_Naped_WStronePoczatku			:= fbCiecie1.fbNaped.PrzesuwanieWStronePoczatku;
stStanyPodzespolow.bCiecie1_Naped_WStroneKonca				:= fbCiecie1.fbNaped.PrzesuwanieWStroneKonca;
stStanyPodzespolow.bCiecie2_Bazowanie						:= fbCiecie2.Bazowanie;
stStanyPodzespolow.bCiecie2_Ciecie							:= fbCiecie2.CyklPracy;
stStanyPodzespolow.bCiecie2_Naped_WStronePoczatku			:= fbCiecie2.fbNaped.PrzesuwanieWStronePoczatku;
stStanyPodzespolow.bCiecie2_Naped_WStroneKonca				:= fbCiecie2.fbNaped.PrzesuwanieWStroneKonca;
stStanyPodzespolow.bPodawanie_Bazowanie						:= fbPodawanieWafla.Bazowanie;
stStanyPodzespolow.bPodawanie_Podawanie						:= fbPodawanieWafla.CyklPracy;
stStanyPodzespolow.bPodawanie_Zabierak_WStronePoczatku		:= fbPodawanieWafla.fbZabierak.PrzesuwanieWStronePoczatku;
stStanyPodzespolow.bPodawanie_zabierak_WStroneKonca			:= fbPodawanieWafla.fbZabierak.PrzesuwanieWStroneKonca;
stStanyPodzespolow.bPodawanie_Przesuwanie_WStronePoczatku	:= fbPodawanieWafla.fbPrzesuwanie.PrzesuwanieWStronePoczatku;
stStanyPodzespolow.bPodawanie_Przesuwanie_WStroneKonca		:= fbPodawanieWafla.fbPrzesuwanie.PrzesuwanieWStroneKonca;
END_METHOD

END_FUNCTION_BLOCK

// ---- POUs/03 - Ciecie/POU/FB_Ciecie.TcPOU
//==================================================================================================
//								RJM Maszyny sp. z o.o.
//									13.05.2022
//	Zespoł siłownika cięcia  
//	Cykl ciecia: ciecie -> odczekanie -> powrot   
// 	v1.0	|| TC v 3.1.4024.22		|| - pierwsza wersja
//==================================================================================================
FUNCTION_BLOCK FB_Ciecie EXTENDS FB_Podzespol
VAR_INPUT
	stParametry								: DUT_Ciecie_Parametry;
END_VAR
VAR_OUTPUT
END_VAR
VAR
	bCzujnik0Naped							: ITF_Czujnik;
	bCzujnikMaxNaped						: ITF_Czujnik;
	fbElektrozaworNaped						: ITF_Elektozawor;
	fbNaped									: FB_Silownik_Kontrola (	fbCzujnikPozycja0 			:= GVL_Wejscia_IO.bCzujnik0C1, 
																		fbCzujnikPozycjaMax 		:= GVL_Wejscia_IO.bCzujnikMaxC1,
																		fbElektrozawor 				:= GVL_Wyjscia_IO.fbElektrozaworC1);

	arrElementyWykonawcze 					: ARRAY [1..GVL_LogowanieBledow_Stale.MAX_ILOSC_ELEMENTOW_NA_PODZESPOL] OF ITF_LogowanieBledow_ElementWykonawczy := 
														[fbNaped.fbLBKomunikacja];
	fbLBKomunikacja							: FB_Ciecie_Komunikacja 
														(arrElementyWykonawcze := arrElementyWykonawcze,
														iIloscPodlementow := 1);		
	tonOdczekaj								: TON;													
END_VAR

METHOD CyklBazowania_Praca : BOOL
VAR_INPUT
END_VAR
IF (NOT bPierwszePrzejscieBazowanie) THEN
	bPierwszePrzejscieBazowanie				:= TRUE;
	bCyklBazowaniaSkonczony					:= FALSE;
	fbNaped.PrzesunDoPoczatku				:= TRUE;
END_IF

IF (fbNaped.NaPoczatku) THEN
	bPierwszePrzejscieBazowanie				:= FALSE;
	bCyklBazowaniaSkonczony					:= TRUE;
	CyklBazowania_Praca						:= FALSE;
ELSE
	CyklBazowania_Praca						:= TRUE;
END_IF
END_METHOD

METHOD CyklPracy_Praca : BOOL
VAR_INPUT
END_VAR
IF (NOT bPierwszePrzejsciePracy) THEN
	bPierwszePrzejsciePracy					:= TRUE;
	bCyklPracySkonczony						:= FALSE;
	fbNaped.PrzesunDoKonca					:= TRUE;
	tonOdczekaj.IN							:= FALSE;
	iKrokPracy								:= 1;
END_IF

CASE iKrokPracy OF
	1	:
	IF (fbNaped.NaKoncu) THEN
		tonOdczekaj.IN						:= TRUE;
		iKrokPracy							:= 10;
	END_IF
	CyklPracy_Praca							:= TRUE;
	10	:
	IF (tonOdczekaj.Q) THEN
		tonOdczekaj.IN						:= FALSE;
		fbNaped.PrzesunDoPoczatku			:= TRUE;
		iKrokPracy							:= 20;
	END_IF
	CyklPracy_Praca							:= TRUE;
	20	:
	IF (fbNaped.NaPoczatku) THEN
		iKrokPracy							:= 30;
	END_IF
	CyklPracy_Praca							:= TRUE;
	30	:
		iKrokPracy							:= 0;
		CyklPracy_Praca						:= FALSE;
END_CASE
END_METHOD

METHOD FB_init : BOOL
VAR_INPUT
	bInitRetains : BOOL; // if TRUE, the retain variables are initialized (warm start / cold start)
	bInCopyCode : BOOL;  // if TRUE, the instance afterwards gets moved into the copy code (online change)
	bCzujnik0Naped							: ITF_Czujnik;
	bCzujnikMaxNaped						: ITF_Czujnik;
	fbElektrozaworNaped						: ITF_Elektozawor;

END_VAR
THIS^.bCzujnik0Naped						:= bCzujnik0Naped;
THIS^.bCzujnikMaxNaped						:= bCzujnikMaxNaped;
THIS^.fbElektrozaworNaped					:= fbElektrozaworNaped;

THIS^.fbNaped.FB_init (FALSE, FALSE, bCzujnik0Naped, bCzujnikMaxNaped, fbElektrozaworNaped);
END_METHOD

PROPERTY Pozycja0 : BOOL
GET
Pozycja0									:= fbNaped.NaPoczatku;
END_GET
END_PROPERTY

